// TIA Portal V17 export
// export: Created 2025-03-10T13:12:59.4902027Z, ExportSetting WithDefaults, DisplayName Totally Integrated Automation Portal, DisplayVersion V17 Update 8, DisplayName TIA Portal Openness, DisplayVersion V17 Update 8, DisplayName TIA Portal Version Control Interface, DisplayVersion V17, DisplayName SINAMICS Startdrive Advanced, DisplayVersion V17 SP2, DisplayName SINAMICS Startdrive G110M, G120, G120C, G120D, G120P, G115D, DisplayVersion V17 SP2, DisplayName SINAMICS Startdrive G130, G150, S120, S150, SINAMICS MV, S210, DisplayVersion V17 SP2, DisplayName STEP 7 Professional, DisplayVersion V17 Update 8, DisplayName SINUMERIK ONE STEP 7 Toolbox, DisplayVersion V17 Update 12, DisplayName SINUMERIK 840D sl STEP 7 Toolbox, DisplayVersion V17 Update 12, DisplayName STEP 7 Safety, DisplayVersion V17 Update 6, DisplayName WinCC Advanced, DisplayVersion V17 Update 8
FUNCTION_BLOCK "FB22702_LOAD_FEEDER_SEQUENCE_WEIGHT"   // FB22702, LAD
TITLE = FB22701 LOAD FEEDER SEQUENCE
{ S7_Optimized_Access := 'FALSE' }
VERSION : 0.1
// stored: AutoNumber false, IsIECCheckEnabled false, SetENOAutomatically false, UDAEnableTagReadback false
   VAR_INPUT
      iCONTROL_ON_DELAYED : Bool;
      iPNEUMATIC_FEEDBACK_ON : Bool;
      iFEEDER_PROFINET_MODE_ACTIVE_FAULT : Bool;
      iFEEDER_LINE_NOT_READY_FAULT : Bool;
      iMOTOR_STIRRER_CONDITIONS : Bool;
      iHOPPER_FEEDBACK_PRESSURE : Real;
      iHOPPER_MOTOR_STIRRER_FEEDBACK_SPEED : Real;
      iPOWDER_FEEDER_HOPPER_FEEDBACK_PRESSURE : Real;
      iHOPPER_WEIGHT_FEEDBACK : Real;
      iTRANSFER_VALVE_FEEDBACK_ON : Bool;
      iTRANSFER_VALVE_FEEDBACK_OFF : Bool;
      iPOWDER_FLOW_ON : Bool;
      iSTART_MANUAL_REQUEST : Bool;
      iSTART_SEMI_REQUEST : Bool;
      iSTART_AUTO_REQUEST : Bool;
      iSTOP_MANUAL_REQUEST : Bool;
      iSTOP_SEMI_REQUEST : Bool;
      iSTOP_AUTO_REQUEST : Bool;
   END_VAR
   VAR_OUTPUT
      oEXCEEDED_TIME_ALARM : Bool;
      oOUT_OF_RANGE_ALARM : Bool;
      oLOST_CONDITIONS : Bool;
      oIS_ALARMS : Bool;
   END_VAR
   VAR_IN_OUT
      MOTOR_STIRRER_SETPOINT : DInt;   // MOTOR STIRRER SETPOINT
      PRESSURE_SETPOINT : Real;   // PRESSURE SETPOINT
   END_VAR
   VAR DB_SPECIFIC
      DATA_SEQUENCE : "GENERAL_DATA_SEQUENCES";
      HMI_STANDARD : "HMI_DATA_START_STOP";
      INPUT_SETTINGS : Struct
         UNIT_NUMBER : Int;
         HOPPER_NUMBER : Int;
      END_STRUCT;
      HMI_SEQUENCE : Struct
         HMI_SEQUENCE_RUNNING : Bool;
         HMI_SEQUENCE_DONE : Bool;
         HMI_SET_KILOGRAMS : UDInt;
         HMI_FEEDBACK_DEPOSITED_KG : UDInt;
         HMI_PRESSURE_INCREMENT : Real;
      END_STRUCT;
      ACTIONS_SEQUENCE : Struct
         REQ_START_TRANSFER_POWDER_VALVE : Bool;   // REQUEST OPEN TRANSFER POWDER VALVE
         REQ_STOP_TRANSFER_POWDER_VALVE : Bool;   // REQUEST CLOSE TRANSFER POWDER VALVE
         REQ_START_PRESSURE_GAS_CONTROL : Bool;   // REQUEST START PRESSURE GAS CONTROL
         REQ_STOP_PRESSURE_GAS_CONTROL : Bool;   // REQUEST STOP PRESSURE GAS CONTROL
         REQ_START_PRESSURE_GAS_VALVE : Bool;   // REQUEST OPEN PRESSURE GAS VALVE
         REQ_STOP_PRESSURE_GAS_VALVE : Bool;   // REQUEST CLOSE PRESSURE GAS VALVE
         REQ_START_RELIEF_GAS_VALVE : Bool;   // REQUEST OPEN RELIEF GAS VALVE
         REQ_STOP_RELIEF_GAS_VALVE : Bool;   // REQUEST CLOSE RELIEF GAS VALVE
         SETPOINT_PRESSURE : Real;   // PRESSURE SETPOINT
         REQUEST_START_MOTOR_STIRRER : Bool;   // REQUEST START MOTOR STIRRER
         REQUEST_STOP_MOTOR_STIRRER : Bool;   // REQUEST STOP MOTOR STIRRER
         SETPOINT_MOTOR_STIRRER : DInt;   // MOTOR STIRRER SETPOINT
      END_STRUCT;
      CONTROL_SEQUENCE : Struct
         HOPPER_PRESSURE_IN_RANGE : Bool;
         HOPPER_MOTOR_STIRRER_IN_RANGE : Bool;
         HOPPER_STIRRER_LOW_RANGE : DInt;
         HOPPER_STIRRER_HIGH_RANGE : DInt;
         HOPPER_PRESSURE_LOW_RANGE : Real;
         HOPPER_PRESSURE_HIGH_RANGE : Real;
         HOPPER_PRESSURE_INCREMENT : Real;
         MATERIAL_APPLIED : Bool;
         WEIGHT_APPLIED : UDInt;
         INITIAL_WEIGHT : Real;
         ESTIMATED_WEIGHT_TO_STOP : Real;
      END_STRUCT;
      INTERNAL : Struct
         TRIGGER_RAISING_EDGE_1 : Bool;
         TRIGGER_RAISING_EDGE_2 : Bool;
         TRIGGER_RAISING_EDGE_3 : Bool;
      END_STRUCT;
      TIMERS : Struct
         TIMER_1 : TON_TIME;
         TIMER_2 : TON_TIME;
         TIMER_3 : TON_TIME;
         TIMER_4 : TON_TIME;
         TIMER_5 : TON_TIME;
         TIMER_6 : TON_TIME;
         TIMER_7 : TON_TIME;
         TIMER_8 : TON_TIME;
         TIMER_9 : TON_TIME;
         TIMER_10 : TON_TIME;
      END_STRUCT;
   END_VAR
   VAR_TEMP
      DB_NUMBER : DInt;
      FEEDER_COVER_PRESSURE_ADDED : Real;
      TIME_EXCEEDED_S5TIME : S5Time;
      TIME_COUNTED : Int;
      TIME_EXCEEDED_TIME : Time;
      TIME_LOAD_IN_MILISEC : Int;
      REMAINING_TIME : Int;
      UINT_TIME_ACTION : UInt;
      LOW_FEEDBACK_PRESSURE : Real;
      HIGH_FEEDBACK_PRESSURE : Real;
      LOW_FEEDBACK_MOTOR_SPEED : Real;
      HIGH_FEEDBACK_MOTOR_SPEED : Real;
   END_VAR
   VAR CONSTANT
      HISTERESIS_PRESSURE : Real := 0.04;
   END_VAR
   // TIMERS.TIMER_1.PT := T#1000ms;
   // TIMERS.TIMER_2.PT := T#1000ms;
   // TIMERS.TIMER_3.PT := T#1000ms;
   // TIMERS.TIMER_4.PT := T#1000ms;
   // TIMERS.TIMER_5.PT := T#1000ms;
   // TIMERS.TIMER_6.PT := T#1000ms;
   // TIMERS.TIMER_7.PT := T#1000ms;
   // TIMERS.TIMER_8.PT := T#1000ms;
   // TIMERS.TIMER_9.PT := T#1000ms;
   VAR_TEMP   // added for the SCL form of the ladder/FBD networks
      _w1 : Bool;
      _w2 : Bool;
   END_VAR
BEGIN

NETWORK
TITLE = READ INSTANCE DB NUMBER
      L     DINO;
      +     10#800000;
      T     #DB_NUMBER;

REGION Network 2: INPUTS
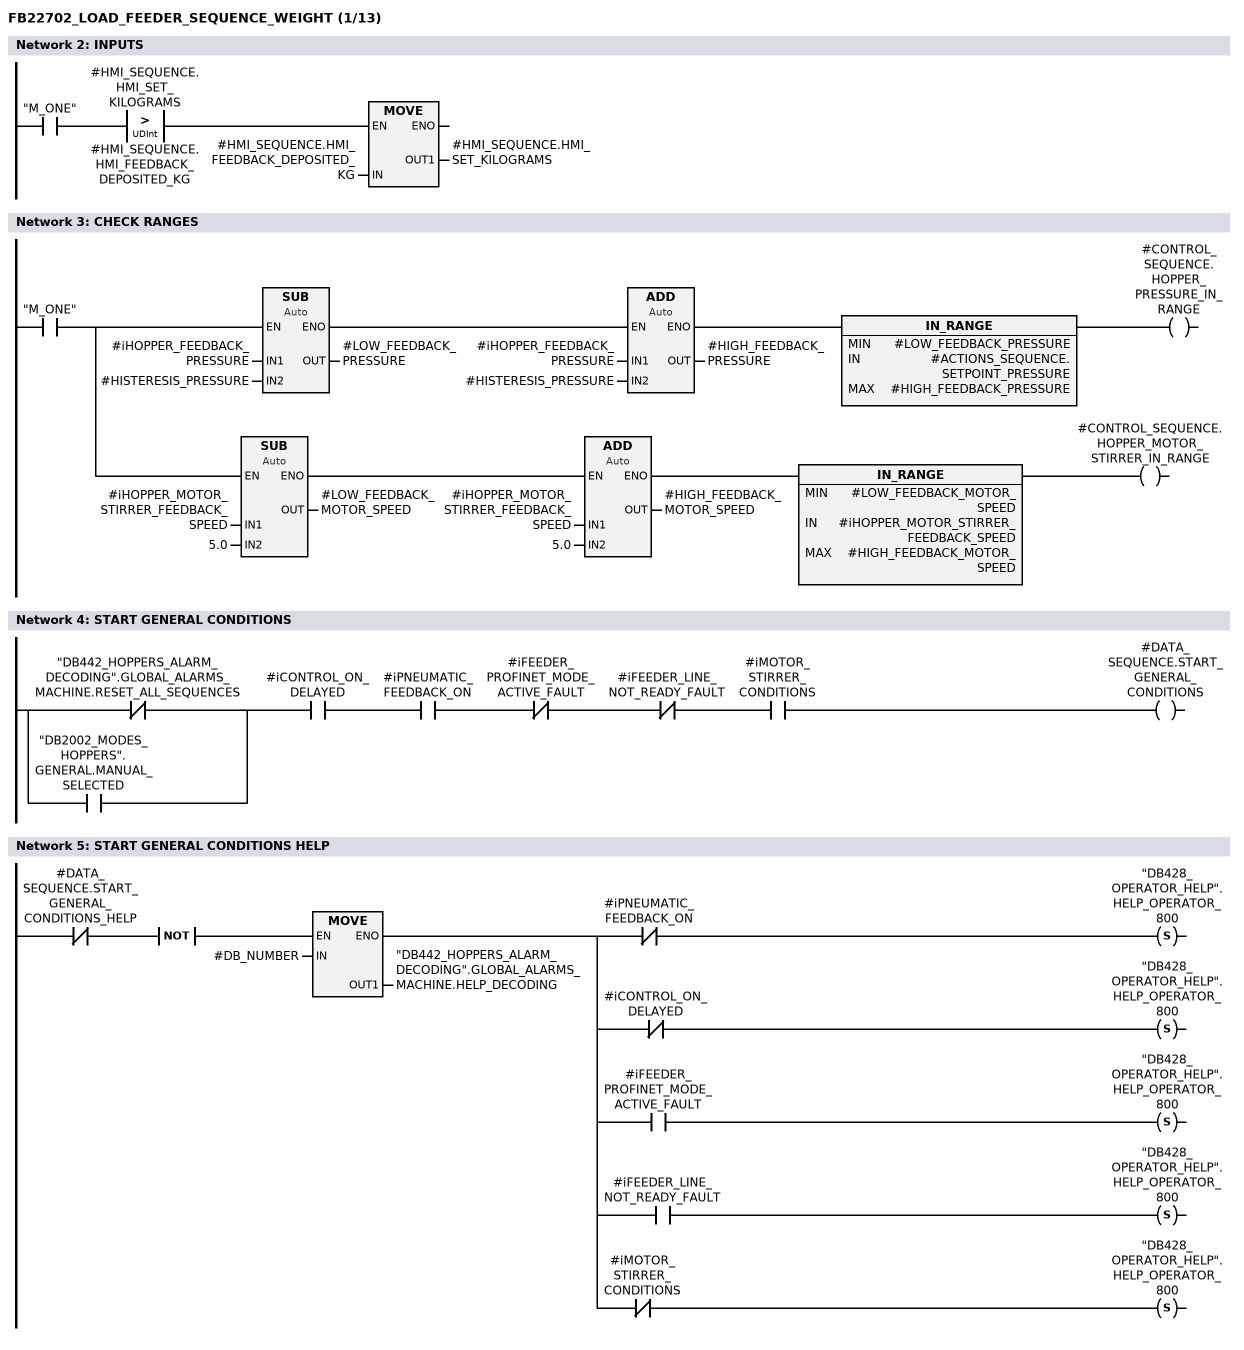
   RUNG wire#powerrail
      Contact( "M_ONE" )
      { S7_Templates := "SrcType := UDInt" } GT_Contact(in1 := #HMI_SEQUENCE.HMI_SET_KILOGRAMS, in2 := #HMI_SEQUENCE.HMI_FEEDBACK_DEPOSITED_KG)
      Move(in := #HMI_SEQUENCE.HMI_FEEDBACK_DEPOSITED_KG, out1 => #HMI_SEQUENCE.HMI_SET_KILOGRAMS)
   END_RUNG
   // the same network as SCL:
   IF "M_ONE" AND (#HMI_SEQUENCE.HMI_SET_KILOGRAMS > #HMI_SEQUENCE.HMI_FEEDBACK_DEPOSITED_KG) THEN
       #HMI_SEQUENCE.HMI_SET_KILOGRAMS := #HMI_SEQUENCE.HMI_FEEDBACK_DEPOSITED_KG;
   END_IF;
END_REGION

REGION Network 3: CHECK RANGES
   RUNG wire#powerrail
      Contact( "M_ONE" )
      wire#w1
      Sub(in1 := #iHOPPER_FEEDBACK_PRESSURE, in2 := #HISTERESIS_PRESSURE, out => #LOW_FEEDBACK_PRESSURE)
      Add(in1 := #iHOPPER_FEEDBACK_PRESSURE, in2 := #HISTERESIS_PRESSURE, out => #HIGH_FEEDBACK_PRESSURE)
      { S7_Templates := "SrcType := Real" } InRange(min := #LOW_FEEDBACK_PRESSURE, in := #ACTIONS_SEQUENCE.SETPOINT_PRESSURE, max := #HIGH_FEEDBACK_PRESSURE)
      Coil( #CONTROL_SEQUENCE.HOPPER_PRESSURE_IN_RANGE )
   END_RUNG
   RUNG wire#w1
      Sub(in1 := #iHOPPER_MOTOR_STIRRER_FEEDBACK_SPEED, in2 := 5.0, out => #LOW_FEEDBACK_MOTOR_SPEED)
      Add(in1 := #iHOPPER_MOTOR_STIRRER_FEEDBACK_SPEED, in2 := 5.0, out => #HIGH_FEEDBACK_MOTOR_SPEED)
      { S7_Templates := "SrcType := Real" } InRange(min := #LOW_FEEDBACK_MOTOR_SPEED, in := #iHOPPER_MOTOR_STIRRER_FEEDBACK_SPEED, max := #HIGH_FEEDBACK_MOTOR_SPEED)
      Coil( #CONTROL_SEQUENCE.HOPPER_MOTOR_STIRRER_IN_RANGE )
   END_RUNG
   // the same network as SCL:
   IF "M_ONE" THEN
       #LOW_FEEDBACK_PRESSURE := #iHOPPER_FEEDBACK_PRESSURE - #HISTERESIS_PRESSURE;
       #HIGH_FEEDBACK_PRESSURE := #iHOPPER_FEEDBACK_PRESSURE + #HISTERESIS_PRESSURE;
   END_IF;
   #CONTROL_SEQUENCE.HOPPER_PRESSURE_IN_RANGE := "M_ONE" AND (#LOW_FEEDBACK_PRESSURE <= #ACTIONS_SEQUENCE.SETPOINT_PRESSURE) AND (#ACTIONS_SEQUENCE.SETPOINT_PRESSURE <= #HIGH_FEEDBACK_PRESSURE);
   IF "M_ONE" THEN
       #LOW_FEEDBACK_MOTOR_SPEED := #iHOPPER_MOTOR_STIRRER_FEEDBACK_SPEED - 5.0;
       #HIGH_FEEDBACK_MOTOR_SPEED := #iHOPPER_MOTOR_STIRRER_FEEDBACK_SPEED + 5.0;
   END_IF;
   #CONTROL_SEQUENCE.HOPPER_MOTOR_STIRRER_IN_RANGE := "M_ONE" AND (#LOW_FEEDBACK_MOTOR_SPEED <= #iHOPPER_MOTOR_STIRRER_FEEDBACK_SPEED) AND (#iHOPPER_MOTOR_STIRRER_FEEDBACK_SPEED <= #HIGH_FEEDBACK_MOTOR_SPEED);
END_REGION

REGION Network 4: START GENERAL CONDITIONS
   RUNG wire#powerrail
      I_Contact( "DB442_HOPPERS_ALARM_DECODING".GLOBAL_ALARMS_MACHINE.RESET_ALL_SEQUENCES )
      wire#w1
      Contact( #iCONTROL_ON_DELAYED )
      Contact( #iPNEUMATIC_FEEDBACK_ON )
      I_Contact( #iFEEDER_PROFINET_MODE_ACTIVE_FAULT )
      I_Contact( #iFEEDER_LINE_NOT_READY_FAULT )
      Contact( #iMOTOR_STIRRER_CONDITIONS )
      Coil( #DATA_SEQUENCE.START_GENERAL_CONDITIONS )
   END_RUNG
   RUNG wire#powerrail
      Contact( "DB2002_MODES_HOPPERS".GENERAL.MANUAL_SELECTED )
   END_RUNG wire#w1
   // the same network as SCL:
   #DATA_SEQUENCE.START_GENERAL_CONDITIONS := (NOT "DB442_HOPPERS_ALARM_DECODING".GLOBAL_ALARMS_MACHINE.RESET_ALL_SEQUENCES OR "DB2002_MODES_HOPPERS".GENERAL.MANUAL_SELECTED) AND #iCONTROL_ON_DELAYED AND #iPNEUMATIC_FEEDBACK_ON AND NOT #iFEEDER_PROFINET_MODE_ACTIVE_FAULT AND NOT #iFEEDER_LINE_NOT_READY_FAULT AND #iMOTOR_STIRRER_CONDITIONS;
END_REGION

REGION Network 5: START GENERAL CONDITIONS HELP
   RUNG wire#powerrail
      I_Contact( #DATA_SEQUENCE.START_GENERAL_CONDITIONS_HELP )
      Not()
      Move(in := #DB_NUMBER, out1 => "DB442_HOPPERS_ALARM_DECODING".GLOBAL_ALARMS_MACHINE.HELP_DECODING)
      wire#w1
      I_Contact( #iPNEUMATIC_FEEDBACK_ON )
      S_Coil( "DB428_OPERATOR_HELP".HELP_OPERATOR_800 )
   END_RUNG
   RUNG wire#w1
      I_Contact( #iCONTROL_ON_DELAYED )
      S_Coil( "DB428_OPERATOR_HELP".HELP_OPERATOR_800 )
   END_RUNG
   RUNG wire#w1
      Contact( #iFEEDER_PROFINET_MODE_ACTIVE_FAULT )
      S_Coil( "DB428_OPERATOR_HELP".HELP_OPERATOR_800 )
   END_RUNG
   RUNG wire#w1
      Contact( #iFEEDER_LINE_NOT_READY_FAULT )
      S_Coil( "DB428_OPERATOR_HELP".HELP_OPERATOR_800 )
   END_RUNG
   RUNG wire#w1
      I_Contact( #iMOTOR_STIRRER_CONDITIONS )
      S_Coil( "DB428_OPERATOR_HELP".HELP_OPERATOR_800 )
   END_RUNG
   // the same network as SCL:
   #_w1 := NOT (NOT #DATA_SEQUENCE.START_GENERAL_CONDITIONS_HELP);
   IF #_w1 THEN "DB442_HOPPERS_ALARM_DECODING".GLOBAL_ALARMS_MACHINE.HELP_DECODING := #DB_NUMBER; END_IF;
   IF #_w1 AND NOT #iPNEUMATIC_FEEDBACK_ON THEN "DB428_OPERATOR_HELP".HELP_OPERATOR_800 := TRUE; END_IF;
   IF #_w1 AND NOT #iCONTROL_ON_DELAYED THEN "DB428_OPERATOR_HELP".HELP_OPERATOR_800 := TRUE; END_IF;
   IF #_w1 AND #iFEEDER_PROFINET_MODE_ACTIVE_FAULT THEN
       "DB428_OPERATOR_HELP".HELP_OPERATOR_800 := TRUE;
   END_IF;
   IF #_w1 AND #iFEEDER_LINE_NOT_READY_FAULT THEN "DB428_OPERATOR_HELP".HELP_OPERATOR_800 := TRUE; END_IF;
   IF #_w1 AND NOT #iMOTOR_STIRRER_CONDITIONS THEN "DB428_OPERATOR_HELP".HELP_OPERATOR_800 := TRUE; END_IF;
END_REGION

REGION Network 6: START INITIAL CONDITIONS / Initial Start Conditions
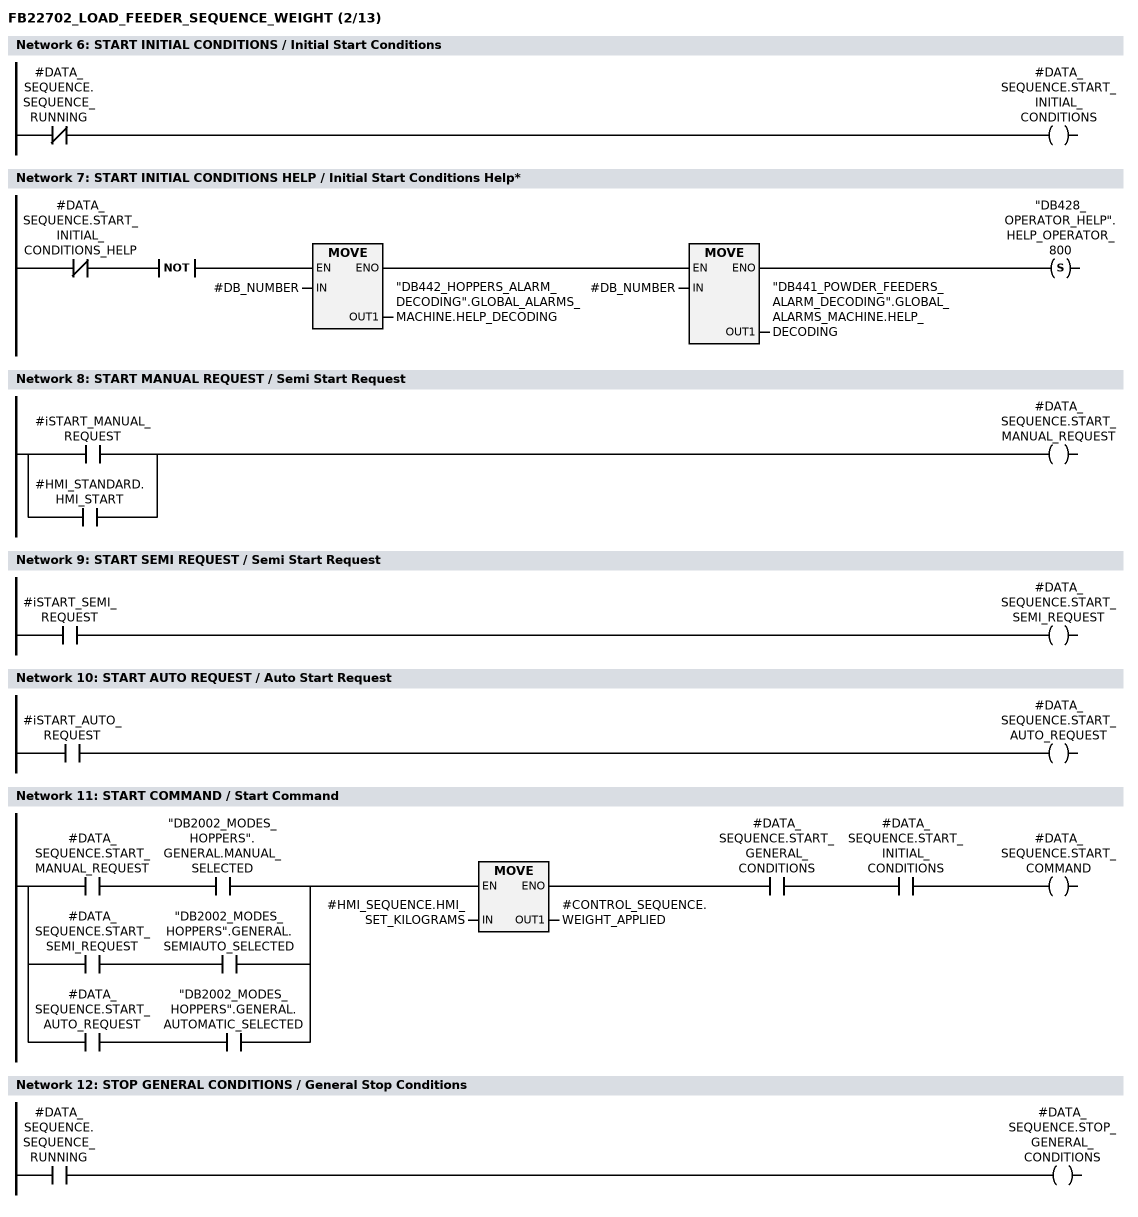
   RUNG wire#powerrail
      I_Contact( #DATA_SEQUENCE.SEQUENCE_RUNNING )
      Coil( #DATA_SEQUENCE.START_INITIAL_CONDITIONS )
   END_RUNG
   // the same network as SCL:
   #DATA_SEQUENCE.START_INITIAL_CONDITIONS := NOT #DATA_SEQUENCE.SEQUENCE_RUNNING;
END_REGION

REGION Network 7: START INITIAL CONDITIONS HELP / Initial Start Conditions Help*
   RUNG wire#powerrail
      I_Contact( #DATA_SEQUENCE.START_INITIAL_CONDITIONS_HELP )
      Not()
      { S7_GenerateENO := "TRUE" } Move(in := #DB_NUMBER, out1 => "DB442_HOPPERS_ALARM_DECODING".GLOBAL_ALARMS_MACHINE.HELP_DECODING)
      { S7_GenerateENO := "TRUE" } Move(in := #DB_NUMBER, out1 => "DB441_POWDER_FEEDERS_ALARM_DECODING".GLOBAL_ALARMS_MACHINE.HELP_DECODING)
      S_Coil( "DB428_OPERATOR_HELP".HELP_OPERATOR_800 )
   END_RUNG
   // the same network as SCL:
   // ENO of a box is taken as its EN; it also drops when the box reports an error
   IF NOT (NOT #DATA_SEQUENCE.START_INITIAL_CONDITIONS_HELP) THEN
       "DB442_HOPPERS_ALARM_DECODING".GLOBAL_ALARMS_MACHINE.HELP_DECODING := #DB_NUMBER;
       "DB441_POWDER_FEEDERS_ALARM_DECODING".GLOBAL_ALARMS_MACHINE.HELP_DECODING := #DB_NUMBER;
       "DB428_OPERATOR_HELP".HELP_OPERATOR_800 := TRUE;
   END_IF;
END_REGION

REGION Network 8: START MANUAL REQUEST / Semi Start Request
   RUNG wire#powerrail
      Contact( #iSTART_MANUAL_REQUEST )
      wire#w1
      Coil( #DATA_SEQUENCE.START_MANUAL_REQUEST )
   END_RUNG
   RUNG wire#powerrail
      Contact( #HMI_STANDARD.HMI_START )
   END_RUNG wire#w1
   // the same network as SCL:
   #DATA_SEQUENCE.START_MANUAL_REQUEST := #iSTART_MANUAL_REQUEST OR #HMI_STANDARD.HMI_START;
END_REGION

REGION Network 9: START SEMI REQUEST / Semi Start Request
   RUNG wire#powerrail
      Contact( #iSTART_SEMI_REQUEST )
      Coil( #DATA_SEQUENCE.START_SEMI_REQUEST )
   END_RUNG
   // the same network as SCL:
   #DATA_SEQUENCE.START_SEMI_REQUEST := #iSTART_SEMI_REQUEST;
END_REGION

REGION Network 10: START AUTO REQUEST / Auto Start Request
   RUNG wire#powerrail
      Contact( #iSTART_AUTO_REQUEST )
      Coil( #DATA_SEQUENCE.START_AUTO_REQUEST )
   END_RUNG
   // the same network as SCL:
   #DATA_SEQUENCE.START_AUTO_REQUEST := #iSTART_AUTO_REQUEST;
END_REGION

REGION Network 11: START COMMAND / Start Command
   RUNG wire#powerrail
      Contact( #DATA_SEQUENCE.START_MANUAL_REQUEST )
      Contact( "DB2002_MODES_HOPPERS".GENERAL.MANUAL_SELECTED )
      wire#w1
      Move(in := #HMI_SEQUENCE.HMI_SET_KILOGRAMS, out1 => #CONTROL_SEQUENCE.WEIGHT_APPLIED)
      Contact( #DATA_SEQUENCE.START_GENERAL_CONDITIONS )
      Contact( #DATA_SEQUENCE.START_INITIAL_CONDITIONS )
      Coil( #DATA_SEQUENCE.START_COMMAND )
   END_RUNG
   RUNG wire#powerrail
      Contact( #DATA_SEQUENCE.START_SEMI_REQUEST )
      Contact( "DB2002_MODES_HOPPERS".GENERAL.SEMIAUTO_SELECTED )
   END_RUNG wire#w1
   RUNG wire#powerrail
      Contact( #DATA_SEQUENCE.START_AUTO_REQUEST )
      Contact( "DB2002_MODES_HOPPERS".GENERAL.AUTOMATIC_SELECTED )
   END_RUNG wire#w1
   // the same network as SCL:
   #_w1 := (#DATA_SEQUENCE.START_MANUAL_REQUEST AND "DB2002_MODES_HOPPERS".GENERAL.MANUAL_SELECTED) OR (#DATA_SEQUENCE.START_SEMI_REQUEST AND "DB2002_MODES_HOPPERS".GENERAL.SEMIAUTO_SELECTED) OR (#DATA_SEQUENCE.START_AUTO_REQUEST AND "DB2002_MODES_HOPPERS".GENERAL.AUTOMATIC_SELECTED);
   IF #_w1 THEN #CONTROL_SEQUENCE.WEIGHT_APPLIED := #HMI_SEQUENCE.HMI_SET_KILOGRAMS; END_IF;
   #DATA_SEQUENCE.START_COMMAND := #_w1 AND #DATA_SEQUENCE.START_GENERAL_CONDITIONS AND #DATA_SEQUENCE.START_INITIAL_CONDITIONS;
END_REGION

REGION Network 12: STOP GENERAL CONDITIONS / General Stop Conditions
   RUNG wire#powerrail
      Contact( #DATA_SEQUENCE.SEQUENCE_RUNNING )
      Coil( #DATA_SEQUENCE.STOP_GENERAL_CONDITIONS )
   END_RUNG
   // the same network as SCL:
   #DATA_SEQUENCE.STOP_GENERAL_CONDITIONS := #DATA_SEQUENCE.SEQUENCE_RUNNING;
END_REGION

REGION Network 13: STOP GENERAL CONDITIONS HELP / General Stop Conditions Help**
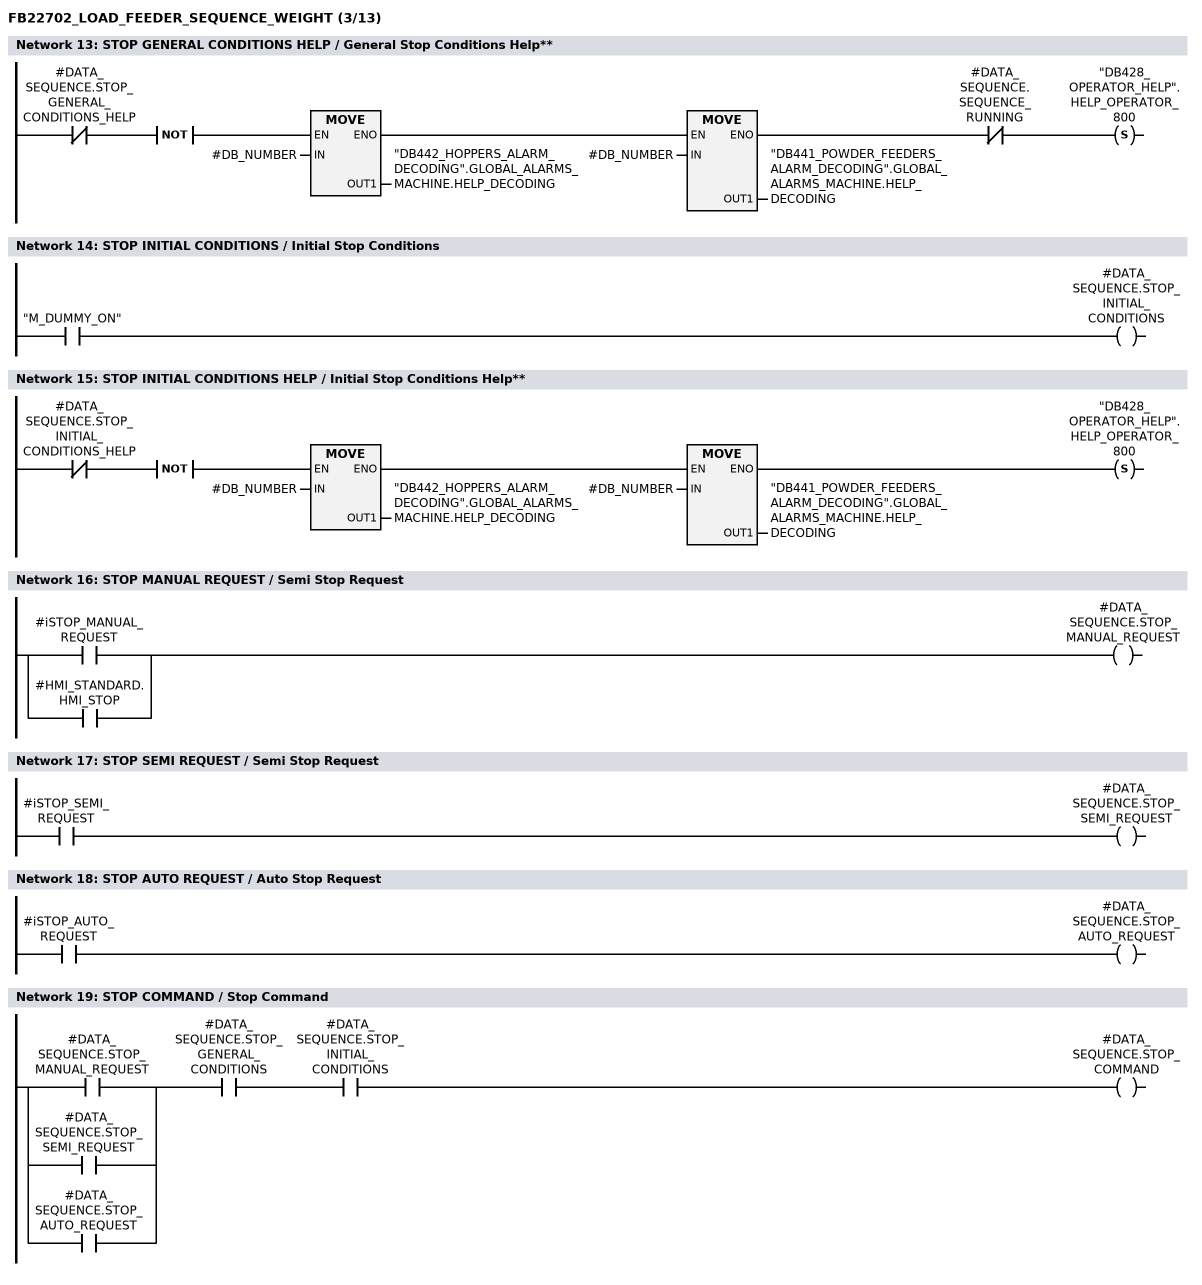
   RUNG wire#powerrail
      I_Contact( #DATA_SEQUENCE.STOP_GENERAL_CONDITIONS_HELP )
      Not()
      { S7_GenerateENO := "TRUE" } Move(in := #DB_NUMBER, out1 => "DB442_HOPPERS_ALARM_DECODING".GLOBAL_ALARMS_MACHINE.HELP_DECODING)
      { S7_GenerateENO := "TRUE" } Move(in := #DB_NUMBER, out1 => "DB441_POWDER_FEEDERS_ALARM_DECODING".GLOBAL_ALARMS_MACHINE.HELP_DECODING)
      I_Contact( #DATA_SEQUENCE.SEQUENCE_RUNNING )
      S_Coil( "DB428_OPERATOR_HELP".HELP_OPERATOR_800 )
   END_RUNG
   // the same network as SCL:
   // ENO of a box is taken as its EN; it also drops when the box reports an error
   #_w1 := NOT (NOT #DATA_SEQUENCE.STOP_GENERAL_CONDITIONS_HELP);
   IF #_w1 THEN
       "DB442_HOPPERS_ALARM_DECODING".GLOBAL_ALARMS_MACHINE.HELP_DECODING := #DB_NUMBER;
       "DB441_POWDER_FEEDERS_ALARM_DECODING".GLOBAL_ALARMS_MACHINE.HELP_DECODING := #DB_NUMBER;
   END_IF;
   IF #_w1 AND NOT #DATA_SEQUENCE.SEQUENCE_RUNNING THEN
       "DB428_OPERATOR_HELP".HELP_OPERATOR_800 := TRUE;
   END_IF;
END_REGION

REGION Network 14: STOP INITIAL CONDITIONS / Initial Stop Conditions
   RUNG wire#powerrail
      Contact( "M_DUMMY_ON" )
      Coil( #DATA_SEQUENCE.STOP_INITIAL_CONDITIONS )
   END_RUNG
   // the same network as SCL:
   #DATA_SEQUENCE.STOP_INITIAL_CONDITIONS := "M_DUMMY_ON";
END_REGION

REGION Network 15: STOP INITIAL CONDITIONS HELP / Initial Stop Conditions Help**
   RUNG wire#powerrail
      I_Contact( #DATA_SEQUENCE.STOP_INITIAL_CONDITIONS_HELP )
      Not()
      { S7_GenerateENO := "TRUE" } Move(in := #DB_NUMBER, out1 => "DB442_HOPPERS_ALARM_DECODING".GLOBAL_ALARMS_MACHINE.HELP_DECODING)
      { S7_GenerateENO := "TRUE" } Move(in := #DB_NUMBER, out1 => "DB441_POWDER_FEEDERS_ALARM_DECODING".GLOBAL_ALARMS_MACHINE.HELP_DECODING)
      S_Coil( "DB428_OPERATOR_HELP".HELP_OPERATOR_800 )
   END_RUNG
   // the same network as SCL:
   // ENO of a box is taken as its EN; it also drops when the box reports an error
   IF NOT (NOT #DATA_SEQUENCE.STOP_INITIAL_CONDITIONS_HELP) THEN
       "DB442_HOPPERS_ALARM_DECODING".GLOBAL_ALARMS_MACHINE.HELP_DECODING := #DB_NUMBER;
       "DB441_POWDER_FEEDERS_ALARM_DECODING".GLOBAL_ALARMS_MACHINE.HELP_DECODING := #DB_NUMBER;
       "DB428_OPERATOR_HELP".HELP_OPERATOR_800 := TRUE;
   END_IF;
END_REGION

REGION Network 16: STOP MANUAL REQUEST / Semi Stop Request
   RUNG wire#powerrail
      Contact( #iSTOP_MANUAL_REQUEST )
      wire#w1
      Coil( #DATA_SEQUENCE.STOP_MANUAL_REQUEST )
   END_RUNG
   RUNG wire#powerrail
      Contact( #HMI_STANDARD.HMI_STOP )
   END_RUNG wire#w1
   // the same network as SCL:
   #DATA_SEQUENCE.STOP_MANUAL_REQUEST := #iSTOP_MANUAL_REQUEST OR #HMI_STANDARD.HMI_STOP;
END_REGION

REGION Network 17: STOP SEMI REQUEST / Semi Stop Request
   RUNG wire#powerrail
      Contact( #iSTOP_SEMI_REQUEST )
      Coil( #DATA_SEQUENCE.STOP_SEMI_REQUEST )
   END_RUNG
   // the same network as SCL:
   #DATA_SEQUENCE.STOP_SEMI_REQUEST := #iSTOP_SEMI_REQUEST;
END_REGION

REGION Network 18: STOP AUTO REQUEST / Auto Stop Request
   RUNG wire#powerrail
      Contact( #iSTOP_AUTO_REQUEST )
      Coil( #DATA_SEQUENCE.STOP_AUTO_REQUEST )
   END_RUNG
   // the same network as SCL:
   #DATA_SEQUENCE.STOP_AUTO_REQUEST := #iSTOP_AUTO_REQUEST;
END_REGION

REGION Network 19: STOP COMMAND / Stop Command
   RUNG wire#powerrail
      Contact( #DATA_SEQUENCE.STOP_MANUAL_REQUEST )
      wire#w1
      Contact( #DATA_SEQUENCE.STOP_GENERAL_CONDITIONS )
      Contact( #DATA_SEQUENCE.STOP_INITIAL_CONDITIONS )
      Coil( #DATA_SEQUENCE.STOP_COMMAND )
   END_RUNG
   RUNG wire#powerrail
      Contact( #DATA_SEQUENCE.STOP_SEMI_REQUEST )
   END_RUNG wire#w1
   RUNG wire#powerrail
      Contact( #DATA_SEQUENCE.STOP_AUTO_REQUEST )
   END_RUNG wire#w1
   // the same network as SCL:
   #DATA_SEQUENCE.STOP_COMMAND := (#DATA_SEQUENCE.STOP_MANUAL_REQUEST OR #DATA_SEQUENCE.STOP_SEMI_REQUEST OR #DATA_SEQUENCE.STOP_AUTO_REQUEST) AND #DATA_SEQUENCE.STOP_GENERAL_CONDITIONS AND #DATA_SEQUENCE.STOP_INITIAL_CONDITIONS;
END_REGION

REGION Network 20: SEQUENCE RUNNING / Sequence Running
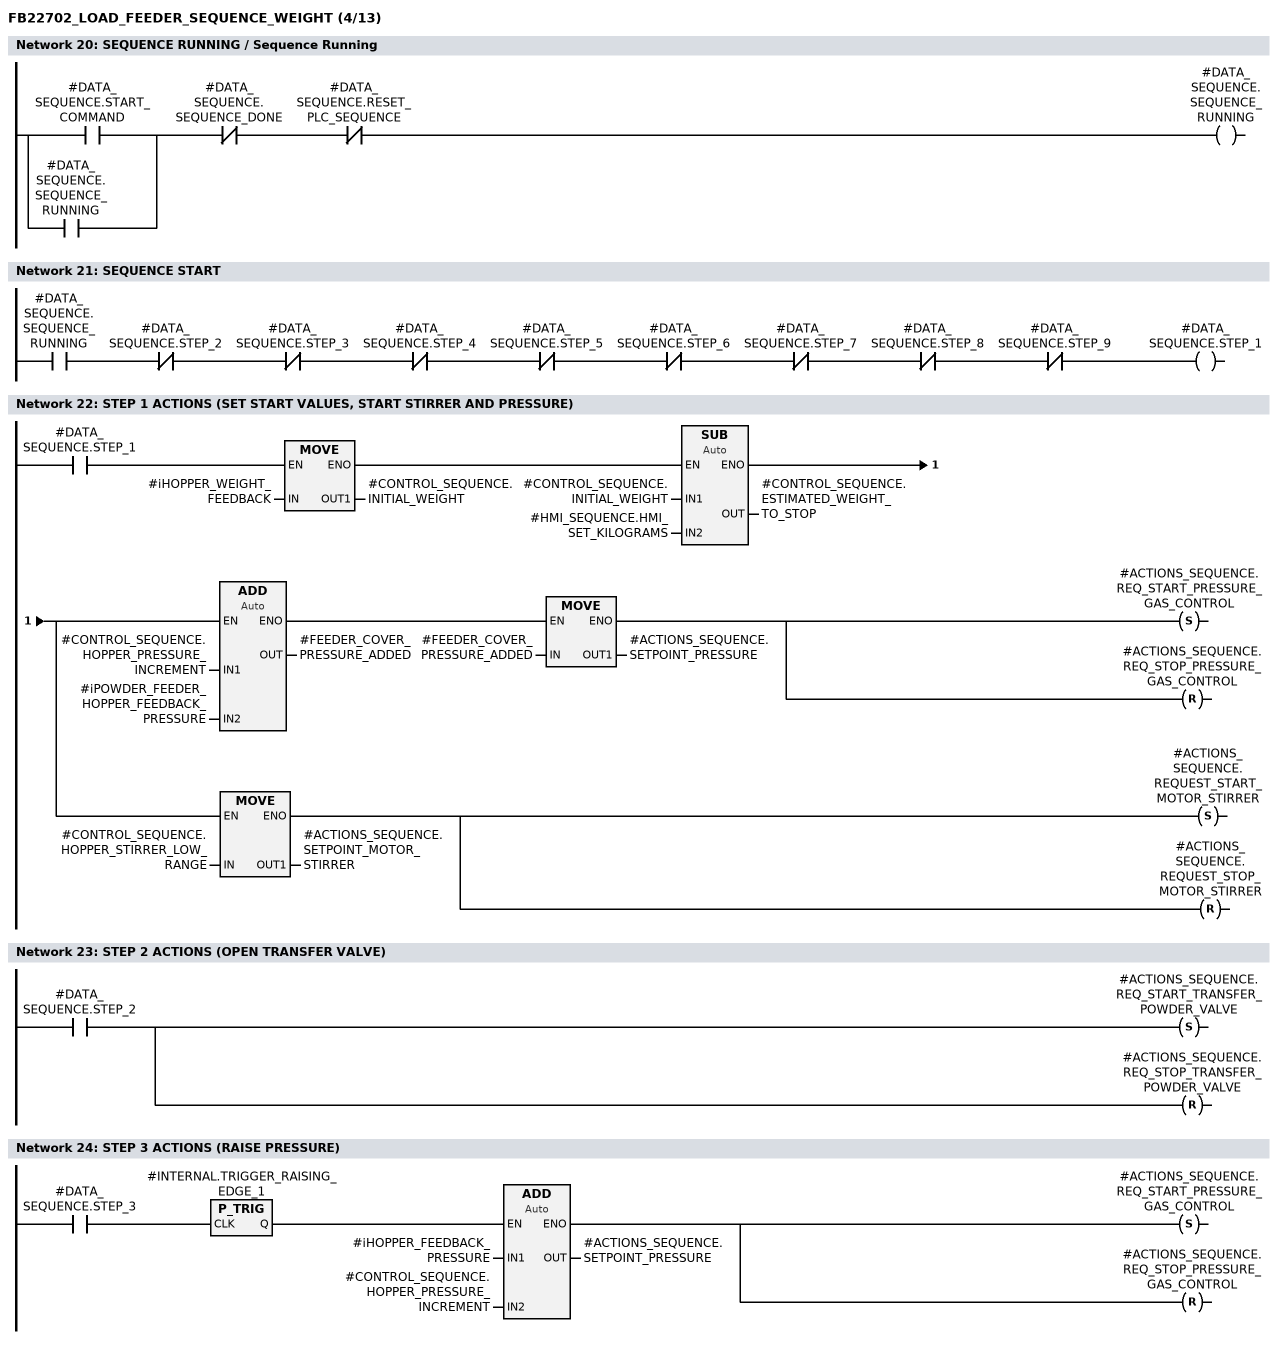
   RUNG wire#powerrail
      Contact( #DATA_SEQUENCE.START_COMMAND )
      wire#w1
      I_Contact( #DATA_SEQUENCE.SEQUENCE_DONE )
      I_Contact( #DATA_SEQUENCE.RESET_PLC_SEQUENCE )
      Coil( #DATA_SEQUENCE.SEQUENCE_RUNNING )
   END_RUNG
   RUNG wire#powerrail
      Contact( #DATA_SEQUENCE.SEQUENCE_RUNNING )
   END_RUNG wire#w1
   // the same network as SCL:
   #DATA_SEQUENCE.SEQUENCE_RUNNING := (#DATA_SEQUENCE.START_COMMAND OR #DATA_SEQUENCE.SEQUENCE_RUNNING) AND NOT #DATA_SEQUENCE.SEQUENCE_DONE AND NOT #DATA_SEQUENCE.RESET_PLC_SEQUENCE;
END_REGION

REGION Network 21: SEQUENCE START
   RUNG wire#powerrail
      Contact( #DATA_SEQUENCE.SEQUENCE_RUNNING )
      I_Contact( #DATA_SEQUENCE.STEP_2 )
      I_Contact( #DATA_SEQUENCE.STEP_3 )
      I_Contact( #DATA_SEQUENCE.STEP_4 )
      I_Contact( #DATA_SEQUENCE.STEP_5 )
      I_Contact( #DATA_SEQUENCE.STEP_6 )
      I_Contact( #DATA_SEQUENCE.STEP_7 )
      I_Contact( #DATA_SEQUENCE.STEP_8 )
      I_Contact( #DATA_SEQUENCE.STEP_9 )
      Coil( #DATA_SEQUENCE.STEP_1 )
   END_RUNG
   // the same network as SCL:
   #DATA_SEQUENCE.STEP_1 := #DATA_SEQUENCE.SEQUENCE_RUNNING AND NOT #DATA_SEQUENCE.STEP_2 AND NOT #DATA_SEQUENCE.STEP_3 AND NOT #DATA_SEQUENCE.STEP_4 AND NOT #DATA_SEQUENCE.STEP_5 AND NOT #DATA_SEQUENCE.STEP_6 AND NOT #DATA_SEQUENCE.STEP_7 AND NOT #DATA_SEQUENCE.STEP_8 AND NOT #DATA_SEQUENCE.STEP_9;
END_REGION

REGION Network 22: STEP 1 ACTIONS (SET START VALUES, START STIRRER AND PRESSURE)
   RUNG wire#powerrail
      Contact( #DATA_SEQUENCE.STEP_1 )
      Move(in := #iHOPPER_WEIGHT_FEEDBACK, out1 => #CONTROL_SEQUENCE.INITIAL_WEIGHT)
      Sub(in1 := #CONTROL_SEQUENCE.INITIAL_WEIGHT, in2 := #HMI_SEQUENCE.HMI_SET_KILOGRAMS, out => #CONTROL_SEQUENCE.ESTIMATED_WEIGHT_TO_STOP)
      wire#w1
      Add(in1 := #CONTROL_SEQUENCE.HOPPER_PRESSURE_INCREMENT, in2 := #iPOWDER_FEEDER_HOPPER_FEEDBACK_PRESSURE, out => #FEEDER_COVER_PRESSURE_ADDED)
      Move(in := #FEEDER_COVER_PRESSURE_ADDED, out1 => #ACTIONS_SEQUENCE.SETPOINT_PRESSURE)
      wire#w2
      S_Coil( #ACTIONS_SEQUENCE.REQ_START_PRESSURE_GAS_CONTROL )
   END_RUNG
   RUNG wire#w2
      R_Coil( #ACTIONS_SEQUENCE.REQ_STOP_PRESSURE_GAS_CONTROL )
   END_RUNG
   RUNG wire#w1
      Move(in := #CONTROL_SEQUENCE.HOPPER_STIRRER_LOW_RANGE, out1 => #ACTIONS_SEQUENCE.SETPOINT_MOTOR_STIRRER)
      wire#w3
      S_Coil( #ACTIONS_SEQUENCE.REQUEST_START_MOTOR_STIRRER )
   END_RUNG
   RUNG wire#w3
      R_Coil( #ACTIONS_SEQUENCE.REQUEST_STOP_MOTOR_STIRRER )
   END_RUNG
   // the same network as SCL:
   IF #DATA_SEQUENCE.STEP_1 THEN
       #CONTROL_SEQUENCE.INITIAL_WEIGHT := #iHOPPER_WEIGHT_FEEDBACK;
       #CONTROL_SEQUENCE.ESTIMATED_WEIGHT_TO_STOP := #CONTROL_SEQUENCE.INITIAL_WEIGHT - #HMI_SEQUENCE.HMI_SET_KILOGRAMS;
       #FEEDER_COVER_PRESSURE_ADDED := #CONTROL_SEQUENCE.HOPPER_PRESSURE_INCREMENT + #iPOWDER_FEEDER_HOPPER_FEEDBACK_PRESSURE;
       #ACTIONS_SEQUENCE.SETPOINT_PRESSURE := #FEEDER_COVER_PRESSURE_ADDED;
       #ACTIONS_SEQUENCE.REQ_START_PRESSURE_GAS_CONTROL := TRUE;
       #ACTIONS_SEQUENCE.REQ_STOP_PRESSURE_GAS_CONTROL := FALSE;
       #ACTIONS_SEQUENCE.SETPOINT_MOTOR_STIRRER := #CONTROL_SEQUENCE.HOPPER_STIRRER_LOW_RANGE;
       #ACTIONS_SEQUENCE.REQUEST_START_MOTOR_STIRRER := TRUE;
       #ACTIONS_SEQUENCE.REQUEST_STOP_MOTOR_STIRRER := FALSE;
   END_IF;
END_REGION

REGION Network 23: STEP 2 ACTIONS (OPEN TRANSFER VALVE)
   RUNG wire#powerrail
      Contact( #DATA_SEQUENCE.STEP_2 )
      wire#w1
      S_Coil( #ACTIONS_SEQUENCE.REQ_START_TRANSFER_POWDER_VALVE )
   END_RUNG
   RUNG wire#w1
      R_Coil( #ACTIONS_SEQUENCE.REQ_STOP_TRANSFER_POWDER_VALVE )
   END_RUNG
   // the same network as SCL:
   IF #DATA_SEQUENCE.STEP_2 THEN
       #ACTIONS_SEQUENCE.REQ_START_TRANSFER_POWDER_VALVE := TRUE;
       #ACTIONS_SEQUENCE.REQ_STOP_TRANSFER_POWDER_VALVE := FALSE;
   END_IF;
END_REGION

REGION Network 24: STEP 3 ACTIONS (RAISE PRESSURE)
   RUNG wire#powerrail
      Contact( #DATA_SEQUENCE.STEP_3 )
      P_Trig( #INTERNAL.TRIGGER_RAISING_EDGE_1 )
      Add(in1 := #iHOPPER_FEEDBACK_PRESSURE, in2 := #CONTROL_SEQUENCE.HOPPER_PRESSURE_INCREMENT, out => #ACTIONS_SEQUENCE.SETPOINT_PRESSURE)
      wire#w1
      S_Coil( #ACTIONS_SEQUENCE.REQ_START_PRESSURE_GAS_CONTROL )
   END_RUNG
   RUNG wire#w1
      R_Coil( #ACTIONS_SEQUENCE.REQ_STOP_PRESSURE_GAS_CONTROL )
   END_RUNG
   // the same network as SCL:
   #_w1 := #DATA_SEQUENCE.STEP_3 AND NOT #INTERNAL.TRIGGER_RAISING_EDGE_1;   // rising edge
   #INTERNAL.TRIGGER_RAISING_EDGE_1 := #DATA_SEQUENCE.STEP_3;
   IF #_w1 THEN
       #ACTIONS_SEQUENCE.SETPOINT_PRESSURE := #iHOPPER_FEEDBACK_PRESSURE + #CONTROL_SEQUENCE.HOPPER_PRESSURE_INCREMENT;
       #ACTIONS_SEQUENCE.REQ_START_PRESSURE_GAS_CONTROL := TRUE;
       #ACTIONS_SEQUENCE.REQ_STOP_PRESSURE_GAS_CONTROL := FALSE;
   END_IF;
END_REGION

REGION Network 25: STEP 4 ACTIONS (RAISE MOTOR SPEED)
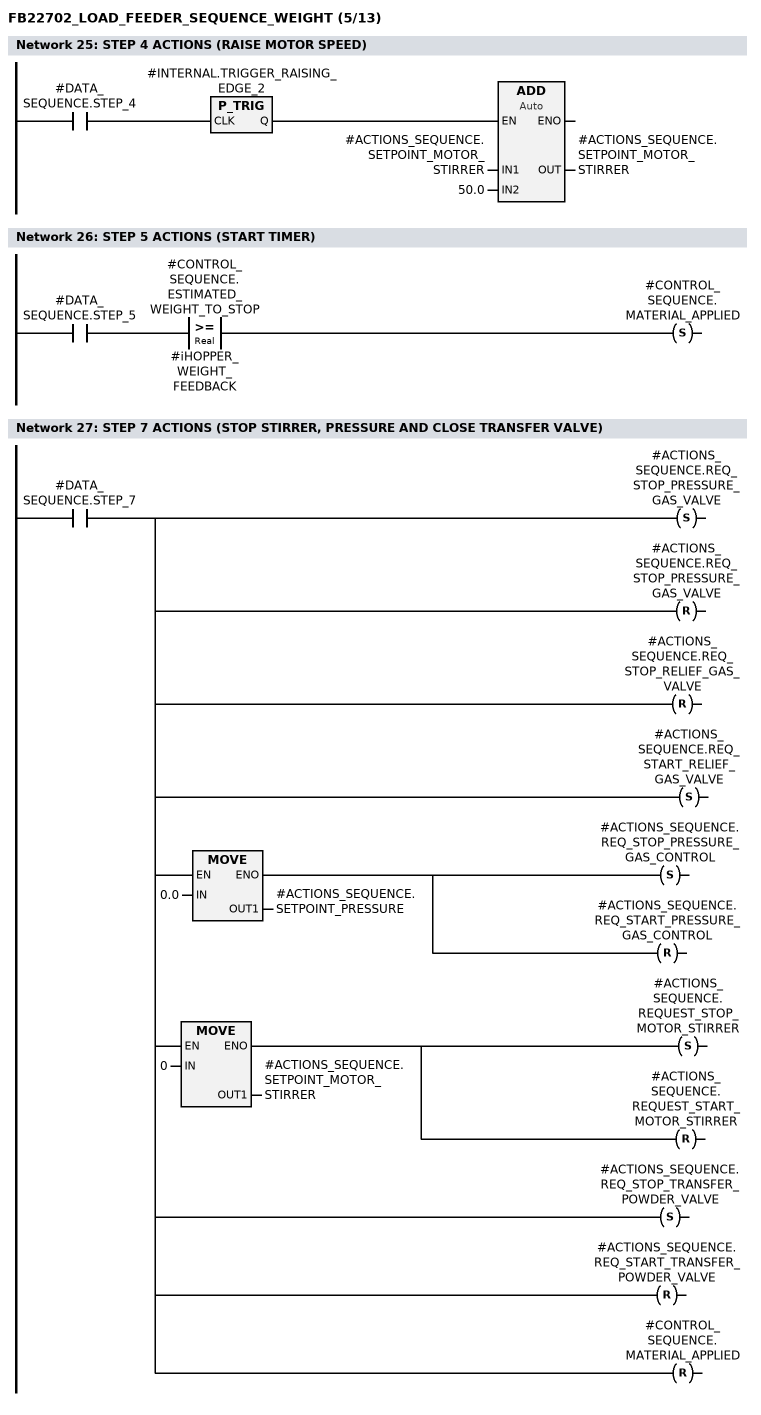
   RUNG wire#powerrail
      Contact( #DATA_SEQUENCE.STEP_4 )
      P_Trig( #INTERNAL.TRIGGER_RAISING_EDGE_2 )
      Add(in1 := #ACTIONS_SEQUENCE.SETPOINT_MOTOR_STIRRER, in2 := 50.0, out => #ACTIONS_SEQUENCE.SETPOINT_MOTOR_STIRRER)
   END_RUNG
   // the same network as SCL:
   #_w1 := #DATA_SEQUENCE.STEP_4 AND NOT #INTERNAL.TRIGGER_RAISING_EDGE_2;   // rising edge
   #INTERNAL.TRIGGER_RAISING_EDGE_2 := #DATA_SEQUENCE.STEP_4;
   IF #_w1 THEN
       #ACTIONS_SEQUENCE.SETPOINT_MOTOR_STIRRER := #ACTIONS_SEQUENCE.SETPOINT_MOTOR_STIRRER + 50.0;
   END_IF;
END_REGION

REGION Network 26: STEP 5 ACTIONS (START TIMER)
   RUNG wire#powerrail
      Contact( #DATA_SEQUENCE.STEP_5 )
      { S7_Templates := "SrcType := Real" } GE_Contact(in1 := #CONTROL_SEQUENCE.ESTIMATED_WEIGHT_TO_STOP, in2 := #iHOPPER_WEIGHT_FEEDBACK)
      S_Coil( #CONTROL_SEQUENCE.MATERIAL_APPLIED )
   END_RUNG
   // the same network as SCL:
   IF #DATA_SEQUENCE.STEP_5 AND (#CONTROL_SEQUENCE.ESTIMATED_WEIGHT_TO_STOP >= #iHOPPER_WEIGHT_FEEDBACK) THEN
       #CONTROL_SEQUENCE.MATERIAL_APPLIED := TRUE;
   END_IF;
END_REGION

REGION Network 27: STEP 7 ACTIONS (STOP STIRRER, PRESSURE AND CLOSE TRANSFER VALVE)
   RUNG wire#powerrail
      Contact( #DATA_SEQUENCE.STEP_7 )
      wire#w1
      S_Coil( #ACTIONS_SEQUENCE.REQ_STOP_PRESSURE_GAS_VALVE )
   END_RUNG
   RUNG wire#w1
      R_Coil( #ACTIONS_SEQUENCE.REQ_STOP_PRESSURE_GAS_VALVE )
   END_RUNG
   RUNG wire#w1
      R_Coil( #ACTIONS_SEQUENCE.REQ_STOP_RELIEF_GAS_VALVE )
   END_RUNG
   RUNG wire#w1
      S_Coil( #ACTIONS_SEQUENCE.REQ_START_RELIEF_GAS_VALVE )
   END_RUNG
   RUNG wire#w1
      Move(in := 0.0, out1 => #ACTIONS_SEQUENCE.SETPOINT_PRESSURE)
      wire#w2
      S_Coil( #ACTIONS_SEQUENCE.REQ_STOP_PRESSURE_GAS_CONTROL )
   END_RUNG
   RUNG wire#w2
      R_Coil( #ACTIONS_SEQUENCE.REQ_START_PRESSURE_GAS_CONTROL )
   END_RUNG
   RUNG wire#w1
      Move(in := 0, out1 => #ACTIONS_SEQUENCE.SETPOINT_MOTOR_STIRRER)
      wire#w3
      S_Coil( #ACTIONS_SEQUENCE.REQUEST_STOP_MOTOR_STIRRER )
   END_RUNG
   RUNG wire#w3
      R_Coil( #ACTIONS_SEQUENCE.REQUEST_START_MOTOR_STIRRER )
   END_RUNG
   RUNG wire#w1
      S_Coil( #ACTIONS_SEQUENCE.REQ_STOP_TRANSFER_POWDER_VALVE )
   END_RUNG
   RUNG wire#w1
      R_Coil( #ACTIONS_SEQUENCE.REQ_START_TRANSFER_POWDER_VALVE )
   END_RUNG
   RUNG wire#w1
      R_Coil( #CONTROL_SEQUENCE.MATERIAL_APPLIED )
   END_RUNG
   // the same network as SCL:
   IF #DATA_SEQUENCE.STEP_7 THEN
       #ACTIONS_SEQUENCE.REQ_STOP_PRESSURE_GAS_VALVE := TRUE;
       #ACTIONS_SEQUENCE.REQ_STOP_PRESSURE_GAS_VALVE := FALSE;
       #ACTIONS_SEQUENCE.REQ_STOP_RELIEF_GAS_VALVE := FALSE;
       #ACTIONS_SEQUENCE.REQ_START_RELIEF_GAS_VALVE := TRUE;
       #ACTIONS_SEQUENCE.SETPOINT_PRESSURE := 0.0;
       #ACTIONS_SEQUENCE.REQ_STOP_PRESSURE_GAS_CONTROL := TRUE;
       #ACTIONS_SEQUENCE.REQ_START_PRESSURE_GAS_CONTROL := FALSE;
       #ACTIONS_SEQUENCE.SETPOINT_MOTOR_STIRRER := 0;
       #ACTIONS_SEQUENCE.REQUEST_STOP_MOTOR_STIRRER := TRUE;
       #ACTIONS_SEQUENCE.REQUEST_START_MOTOR_STIRRER := FALSE;
       #ACTIONS_SEQUENCE.REQ_STOP_TRANSFER_POWDER_VALVE := TRUE;
       #ACTIONS_SEQUENCE.REQ_START_TRANSFER_POWDER_VALVE := FALSE;
       #CONTROL_SEQUENCE.MATERIAL_APPLIED := FALSE;
   END_IF;
END_REGION

REGION Network 28: STEP 8 ACTIONS(STOP STIRRER, PRESSURE AND CLOSE TRANSFER VALVE)
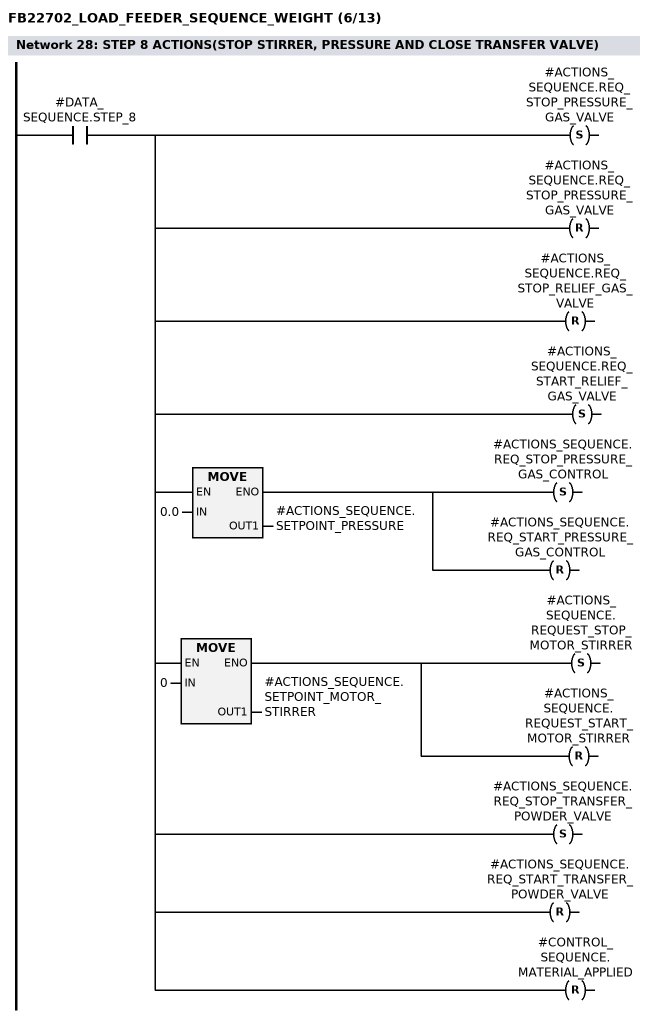
   RUNG wire#powerrail
      Contact( #DATA_SEQUENCE.STEP_8 )
      wire#w1
      S_Coil( #ACTIONS_SEQUENCE.REQ_STOP_PRESSURE_GAS_VALVE )
   END_RUNG
   RUNG wire#w1
      R_Coil( #ACTIONS_SEQUENCE.REQ_STOP_PRESSURE_GAS_VALVE )
   END_RUNG
   RUNG wire#w1
      R_Coil( #ACTIONS_SEQUENCE.REQ_STOP_RELIEF_GAS_VALVE )
   END_RUNG
   RUNG wire#w1
      S_Coil( #ACTIONS_SEQUENCE.REQ_START_RELIEF_GAS_VALVE )
   END_RUNG
   RUNG wire#w1
      Move(in := 0.0, out1 => #ACTIONS_SEQUENCE.SETPOINT_PRESSURE)
      wire#w2
      S_Coil( #ACTIONS_SEQUENCE.REQ_STOP_PRESSURE_GAS_CONTROL )
   END_RUNG
   RUNG wire#w2
      R_Coil( #ACTIONS_SEQUENCE.REQ_START_PRESSURE_GAS_CONTROL )
   END_RUNG
   RUNG wire#w1
      Move(in := 0, out1 => #ACTIONS_SEQUENCE.SETPOINT_MOTOR_STIRRER)
      wire#w3
      S_Coil( #ACTIONS_SEQUENCE.REQUEST_STOP_MOTOR_STIRRER )
   END_RUNG
   RUNG wire#w3
      R_Coil( #ACTIONS_SEQUENCE.REQUEST_START_MOTOR_STIRRER )
   END_RUNG
   RUNG wire#w1
      S_Coil( #ACTIONS_SEQUENCE.REQ_STOP_TRANSFER_POWDER_VALVE )
   END_RUNG
   RUNG wire#w1
      R_Coil( #ACTIONS_SEQUENCE.REQ_START_TRANSFER_POWDER_VALVE )
   END_RUNG
   RUNG wire#w1
      R_Coil( #CONTROL_SEQUENCE.MATERIAL_APPLIED )
   END_RUNG
   // the same network as SCL:
   IF #DATA_SEQUENCE.STEP_8 THEN
       #ACTIONS_SEQUENCE.REQ_STOP_PRESSURE_GAS_VALVE := TRUE;
       #ACTIONS_SEQUENCE.REQ_STOP_PRESSURE_GAS_VALVE := FALSE;
       #ACTIONS_SEQUENCE.REQ_STOP_RELIEF_GAS_VALVE := FALSE;
       #ACTIONS_SEQUENCE.REQ_START_RELIEF_GAS_VALVE := TRUE;
       #ACTIONS_SEQUENCE.SETPOINT_PRESSURE := 0.0;
       #ACTIONS_SEQUENCE.REQ_STOP_PRESSURE_GAS_CONTROL := TRUE;
       #ACTIONS_SEQUENCE.REQ_START_PRESSURE_GAS_CONTROL := FALSE;
       #ACTIONS_SEQUENCE.SETPOINT_MOTOR_STIRRER := 0;
       #ACTIONS_SEQUENCE.REQUEST_STOP_MOTOR_STIRRER := TRUE;
       #ACTIONS_SEQUENCE.REQUEST_START_MOTOR_STIRRER := FALSE;
       #ACTIONS_SEQUENCE.REQ_STOP_TRANSFER_POWDER_VALVE := TRUE;
       #ACTIONS_SEQUENCE.REQ_START_TRANSFER_POWDER_VALVE := FALSE;
       #CONTROL_SEQUENCE.MATERIAL_APPLIED := FALSE;
   END_IF;
END_REGION

REGION Network 29: STEP 9 ACTIONS (RESET VARIABLES)
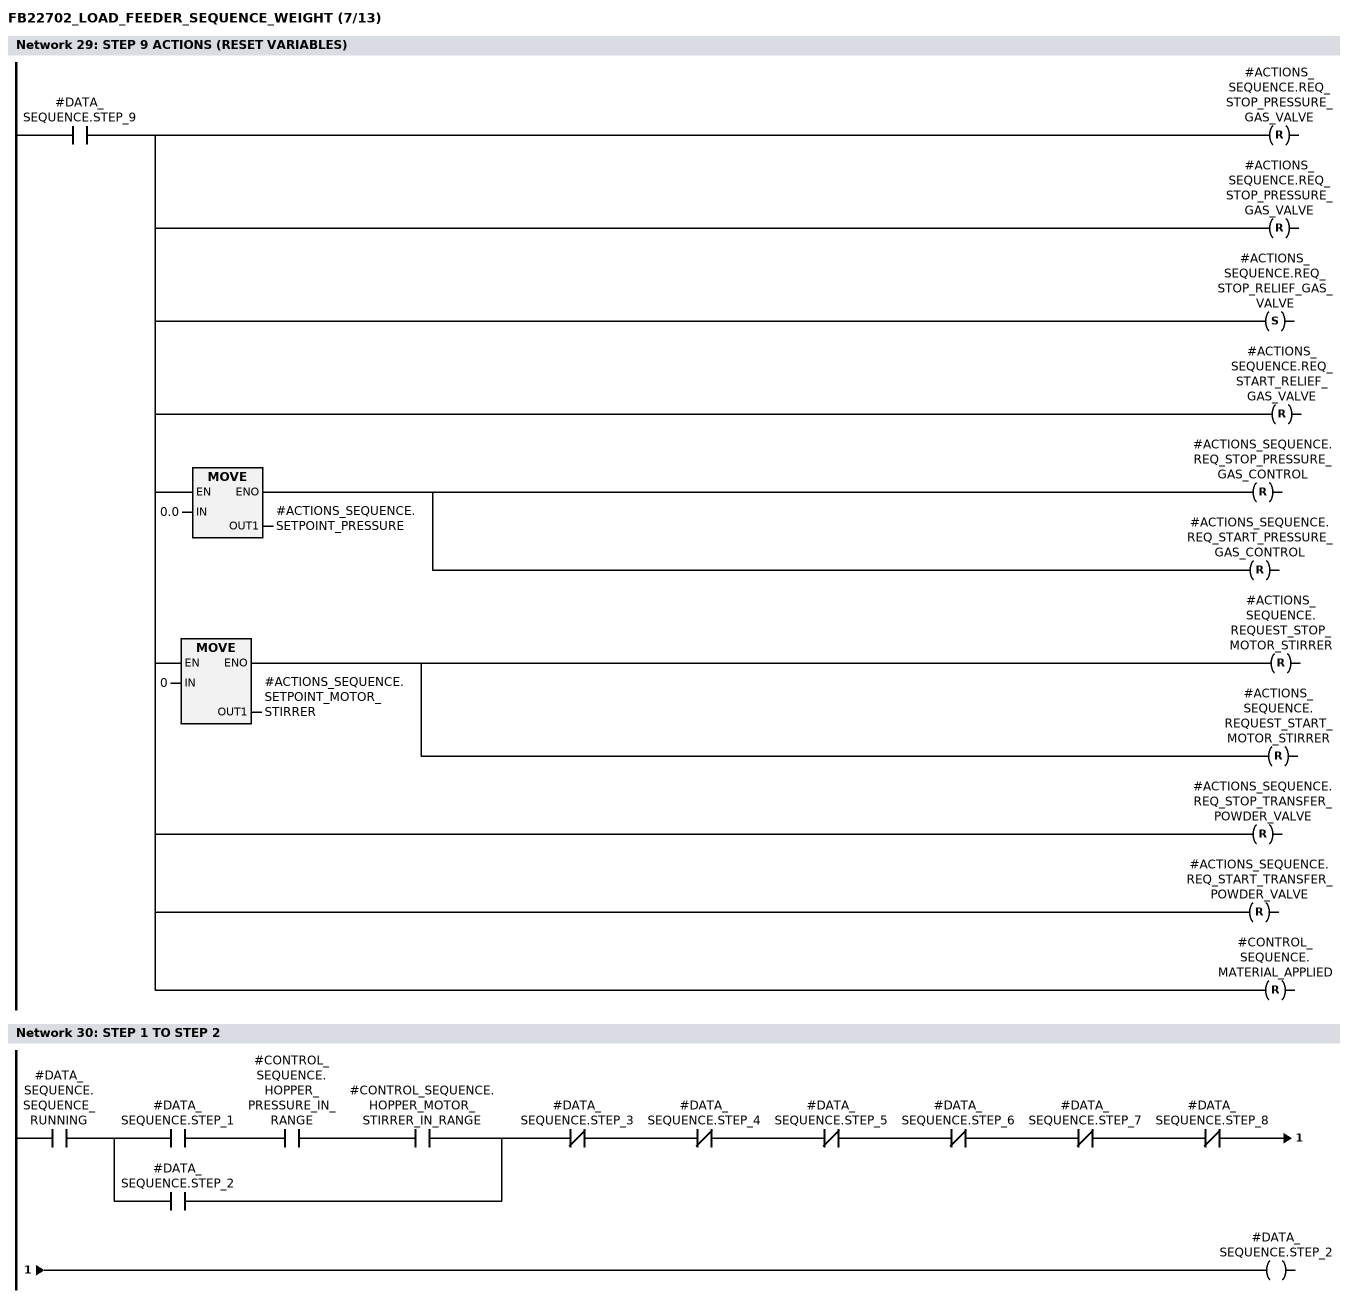
   RUNG wire#powerrail
      Contact( #DATA_SEQUENCE.STEP_9 )
      wire#w1
      R_Coil( #ACTIONS_SEQUENCE.REQ_STOP_PRESSURE_GAS_VALVE )
   END_RUNG
   RUNG wire#w1
      R_Coil( #ACTIONS_SEQUENCE.REQ_STOP_PRESSURE_GAS_VALVE )
   END_RUNG
   RUNG wire#w1
      S_Coil( #ACTIONS_SEQUENCE.REQ_STOP_RELIEF_GAS_VALVE )
   END_RUNG
   RUNG wire#w1
      R_Coil( #ACTIONS_SEQUENCE.REQ_START_RELIEF_GAS_VALVE )
   END_RUNG
   RUNG wire#w1
      Move(in := 0.0, out1 => #ACTIONS_SEQUENCE.SETPOINT_PRESSURE)
      wire#w2
      R_Coil( #ACTIONS_SEQUENCE.REQ_STOP_PRESSURE_GAS_CONTROL )
   END_RUNG
   RUNG wire#w2
      R_Coil( #ACTIONS_SEQUENCE.REQ_START_PRESSURE_GAS_CONTROL )
   END_RUNG
   RUNG wire#w1
      Move(in := 0, out1 => #ACTIONS_SEQUENCE.SETPOINT_MOTOR_STIRRER)
      wire#w3
      R_Coil( #ACTIONS_SEQUENCE.REQUEST_STOP_MOTOR_STIRRER )
   END_RUNG
   RUNG wire#w3
      R_Coil( #ACTIONS_SEQUENCE.REQUEST_START_MOTOR_STIRRER )
   END_RUNG
   RUNG wire#w1
      R_Coil( #ACTIONS_SEQUENCE.REQ_STOP_TRANSFER_POWDER_VALVE )
   END_RUNG
   RUNG wire#w1
      R_Coil( #ACTIONS_SEQUENCE.REQ_START_TRANSFER_POWDER_VALVE )
   END_RUNG
   RUNG wire#w1
      R_Coil( #CONTROL_SEQUENCE.MATERIAL_APPLIED )
   END_RUNG
   // the same network as SCL:
   IF #DATA_SEQUENCE.STEP_9 THEN
       #ACTIONS_SEQUENCE.REQ_STOP_PRESSURE_GAS_VALVE := FALSE;
       #ACTIONS_SEQUENCE.REQ_STOP_PRESSURE_GAS_VALVE := FALSE;
       #ACTIONS_SEQUENCE.REQ_STOP_RELIEF_GAS_VALVE := TRUE;
       #ACTIONS_SEQUENCE.REQ_START_RELIEF_GAS_VALVE := FALSE;
       #ACTIONS_SEQUENCE.SETPOINT_PRESSURE := 0.0;
       #ACTIONS_SEQUENCE.REQ_STOP_PRESSURE_GAS_CONTROL := FALSE;
       #ACTIONS_SEQUENCE.REQ_START_PRESSURE_GAS_CONTROL := FALSE;
       #ACTIONS_SEQUENCE.SETPOINT_MOTOR_STIRRER := 0;
       #ACTIONS_SEQUENCE.REQUEST_STOP_MOTOR_STIRRER := FALSE;
       #ACTIONS_SEQUENCE.REQUEST_START_MOTOR_STIRRER := FALSE;
       #ACTIONS_SEQUENCE.REQ_STOP_TRANSFER_POWDER_VALVE := FALSE;
       #ACTIONS_SEQUENCE.REQ_START_TRANSFER_POWDER_VALVE := FALSE;
       #CONTROL_SEQUENCE.MATERIAL_APPLIED := FALSE;
   END_IF;
END_REGION

REGION Network 30: STEP 1 TO STEP 2
   RUNG wire#powerrail
      Contact( #DATA_SEQUENCE.SEQUENCE_RUNNING )
      wire#w1
      Contact( #DATA_SEQUENCE.STEP_1 )
      Contact( #CONTROL_SEQUENCE.HOPPER_PRESSURE_IN_RANGE )
      Contact( #CONTROL_SEQUENCE.HOPPER_MOTOR_STIRRER_IN_RANGE )
      wire#w2
      I_Contact( #DATA_SEQUENCE.STEP_3 )
      I_Contact( #DATA_SEQUENCE.STEP_4 )
      I_Contact( #DATA_SEQUENCE.STEP_5 )
      I_Contact( #DATA_SEQUENCE.STEP_6 )
      I_Contact( #DATA_SEQUENCE.STEP_7 )
      I_Contact( #DATA_SEQUENCE.STEP_8 )
      Coil( #DATA_SEQUENCE.STEP_2 )
   END_RUNG
   RUNG wire#w1
      Contact( #DATA_SEQUENCE.STEP_2 )
   END_RUNG wire#w2
   // the same network as SCL:
   #DATA_SEQUENCE.STEP_2 := #DATA_SEQUENCE.SEQUENCE_RUNNING AND ((#DATA_SEQUENCE.STEP_1 AND #CONTROL_SEQUENCE.HOPPER_PRESSURE_IN_RANGE AND #CONTROL_SEQUENCE.HOPPER_MOTOR_STIRRER_IN_RANGE) OR #DATA_SEQUENCE.STEP_2) AND NOT #DATA_SEQUENCE.STEP_3 AND NOT #DATA_SEQUENCE.STEP_4 AND NOT #DATA_SEQUENCE.STEP_5 AND NOT #DATA_SEQUENCE.STEP_6 AND NOT #DATA_SEQUENCE.STEP_7 AND NOT #DATA_SEQUENCE.STEP_8;
END_REGION

REGION Network 31: STEP 2, 6, 4 TO STEP 3
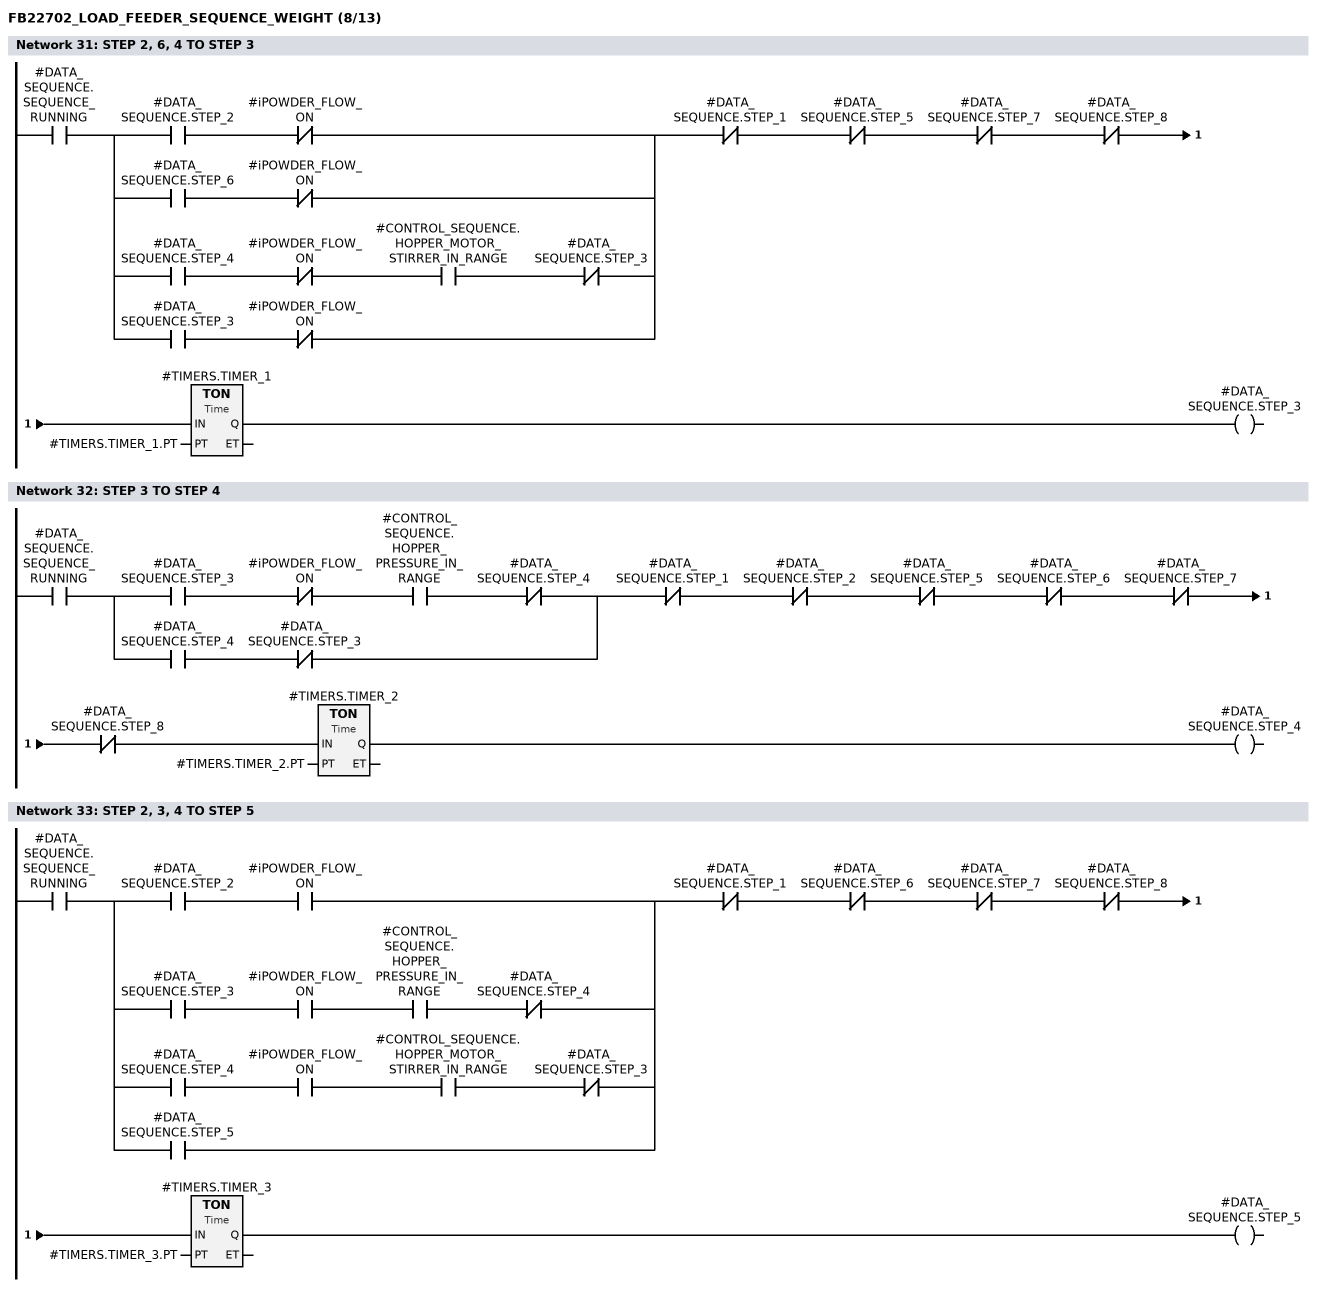
   RUNG wire#powerrail
      Contact( #DATA_SEQUENCE.SEQUENCE_RUNNING )
      wire#w1
      Contact( #DATA_SEQUENCE.STEP_2 )
      I_Contact( #iPOWDER_FLOW_ON )
      wire#w2
      I_Contact( #DATA_SEQUENCE.STEP_1 )
      I_Contact( #DATA_SEQUENCE.STEP_5 )
      I_Contact( #DATA_SEQUENCE.STEP_7 )
      I_Contact( #DATA_SEQUENCE.STEP_8 )
      { S7_Templates := "time_type := Time" } #TIMERS.TIMER_1.TON(pt := #TIMERS.TIMER_1.PT, et =>)
      Coil( #DATA_SEQUENCE.STEP_3 )
   END_RUNG
   RUNG wire#w1
      Contact( #DATA_SEQUENCE.STEP_6 )
      I_Contact( #iPOWDER_FLOW_ON )
   END_RUNG wire#w2
   RUNG wire#w1
      Contact( #DATA_SEQUENCE.STEP_4 )
      I_Contact( #iPOWDER_FLOW_ON )
      Contact( #CONTROL_SEQUENCE.HOPPER_MOTOR_STIRRER_IN_RANGE )
      I_Contact( #DATA_SEQUENCE.STEP_3 )
   END_RUNG wire#w2
   RUNG wire#w1
      Contact( #DATA_SEQUENCE.STEP_3 )
      I_Contact( #iPOWDER_FLOW_ON )
   END_RUNG wire#w2
   // the same network as SCL:
   #TIMERS.TIMER_1.TON(IN := #DATA_SEQUENCE.SEQUENCE_RUNNING AND ((#DATA_SEQUENCE.STEP_2 AND NOT #iPOWDER_FLOW_ON) OR (#DATA_SEQUENCE.STEP_6 AND NOT #iPOWDER_FLOW_ON) OR (#DATA_SEQUENCE.STEP_4 AND NOT #iPOWDER_FLOW_ON AND #CONTROL_SEQUENCE.HOPPER_MOTOR_STIRRER_IN_RANGE AND NOT #DATA_SEQUENCE.STEP_3) OR (#DATA_SEQUENCE.STEP_3 AND NOT #iPOWDER_FLOW_ON)) AND NOT #DATA_SEQUENCE.STEP_1 AND NOT #DATA_SEQUENCE.STEP_5 AND NOT #DATA_SEQUENCE.STEP_7 AND NOT #DATA_SEQUENCE.STEP_8,
                       PT := #TIMERS.TIMER_1.PT);
   #DATA_SEQUENCE.STEP_3 := #TIMERS.TIMER_1.Q;
END_REGION

REGION Network 32: STEP 3 TO STEP 4
   RUNG wire#powerrail
      Contact( #DATA_SEQUENCE.SEQUENCE_RUNNING )
      wire#w1
      Contact( #DATA_SEQUENCE.STEP_3 )
      I_Contact( #iPOWDER_FLOW_ON )
      Contact( #CONTROL_SEQUENCE.HOPPER_PRESSURE_IN_RANGE )
      I_Contact( #DATA_SEQUENCE.STEP_4 )
      wire#w2
      I_Contact( #DATA_SEQUENCE.STEP_1 )
      I_Contact( #DATA_SEQUENCE.STEP_2 )
      I_Contact( #DATA_SEQUENCE.STEP_5 )
      I_Contact( #DATA_SEQUENCE.STEP_6 )
      I_Contact( #DATA_SEQUENCE.STEP_7 )
      I_Contact( #DATA_SEQUENCE.STEP_8 )
      { S7_Templates := "time_type := Time" } #TIMERS.TIMER_2.TON(pt := #TIMERS.TIMER_2.PT, et =>)
      Coil( #DATA_SEQUENCE.STEP_4 )
   END_RUNG
   RUNG wire#w1
      Contact( #DATA_SEQUENCE.STEP_4 )
      I_Contact( #DATA_SEQUENCE.STEP_3 )
   END_RUNG wire#w2
   // the same network as SCL:
   #TIMERS.TIMER_2.TON(IN := #DATA_SEQUENCE.SEQUENCE_RUNNING AND ((#DATA_SEQUENCE.STEP_3 AND NOT #iPOWDER_FLOW_ON AND #CONTROL_SEQUENCE.HOPPER_PRESSURE_IN_RANGE AND NOT #DATA_SEQUENCE.STEP_4) OR (#DATA_SEQUENCE.STEP_4 AND NOT #DATA_SEQUENCE.STEP_3)) AND NOT #DATA_SEQUENCE.STEP_1 AND NOT #DATA_SEQUENCE.STEP_2 AND NOT #DATA_SEQUENCE.STEP_5 AND NOT #DATA_SEQUENCE.STEP_6 AND NOT #DATA_SEQUENCE.STEP_7 AND NOT #DATA_SEQUENCE.STEP_8,
                       PT := #TIMERS.TIMER_2.PT);
   #DATA_SEQUENCE.STEP_4 := #TIMERS.TIMER_2.Q;
END_REGION

REGION Network 33: STEP 2, 3, 4 TO STEP 5
   RUNG wire#powerrail
      Contact( #DATA_SEQUENCE.SEQUENCE_RUNNING )
      wire#w1
      Contact( #DATA_SEQUENCE.STEP_2 )
      Contact( #iPOWDER_FLOW_ON )
      wire#w2
      I_Contact( #DATA_SEQUENCE.STEP_1 )
      I_Contact( #DATA_SEQUENCE.STEP_6 )
      I_Contact( #DATA_SEQUENCE.STEP_7 )
      I_Contact( #DATA_SEQUENCE.STEP_8 )
      { S7_Templates := "time_type := Time" } #TIMERS.TIMER_3.TON(pt := #TIMERS.TIMER_3.PT, et =>)
      Coil( #DATA_SEQUENCE.STEP_5 )
   END_RUNG
   RUNG wire#w1
      Contact( #DATA_SEQUENCE.STEP_3 )
      Contact( #iPOWDER_FLOW_ON )
      Contact( #CONTROL_SEQUENCE.HOPPER_PRESSURE_IN_RANGE )
      I_Contact( #DATA_SEQUENCE.STEP_4 )
   END_RUNG wire#w2
   RUNG wire#w1
      Contact( #DATA_SEQUENCE.STEP_4 )
      Contact( #iPOWDER_FLOW_ON )
      Contact( #CONTROL_SEQUENCE.HOPPER_MOTOR_STIRRER_IN_RANGE )
      I_Contact( #DATA_SEQUENCE.STEP_3 )
   END_RUNG wire#w2
   RUNG wire#w1
      Contact( #DATA_SEQUENCE.STEP_5 )
   END_RUNG wire#w2
   // the same network as SCL:
   #TIMERS.TIMER_3.TON(IN := #DATA_SEQUENCE.SEQUENCE_RUNNING AND ((#DATA_SEQUENCE.STEP_2 AND #iPOWDER_FLOW_ON) OR (#DATA_SEQUENCE.STEP_3 AND #iPOWDER_FLOW_ON AND #CONTROL_SEQUENCE.HOPPER_PRESSURE_IN_RANGE AND NOT #DATA_SEQUENCE.STEP_4) OR (#DATA_SEQUENCE.STEP_4 AND #iPOWDER_FLOW_ON AND #CONTROL_SEQUENCE.HOPPER_MOTOR_STIRRER_IN_RANGE AND NOT #DATA_SEQUENCE.STEP_3) OR #DATA_SEQUENCE.STEP_5) AND NOT #DATA_SEQUENCE.STEP_1 AND NOT #DATA_SEQUENCE.STEP_6 AND NOT #DATA_SEQUENCE.STEP_7 AND NOT #DATA_SEQUENCE.STEP_8,
                       PT := #TIMERS.TIMER_3.PT);
   #DATA_SEQUENCE.STEP_5 := #TIMERS.TIMER_3.Q;
END_REGION

REGION Network 34: STEP 5 AND STOP COMMAND TO STEP 7
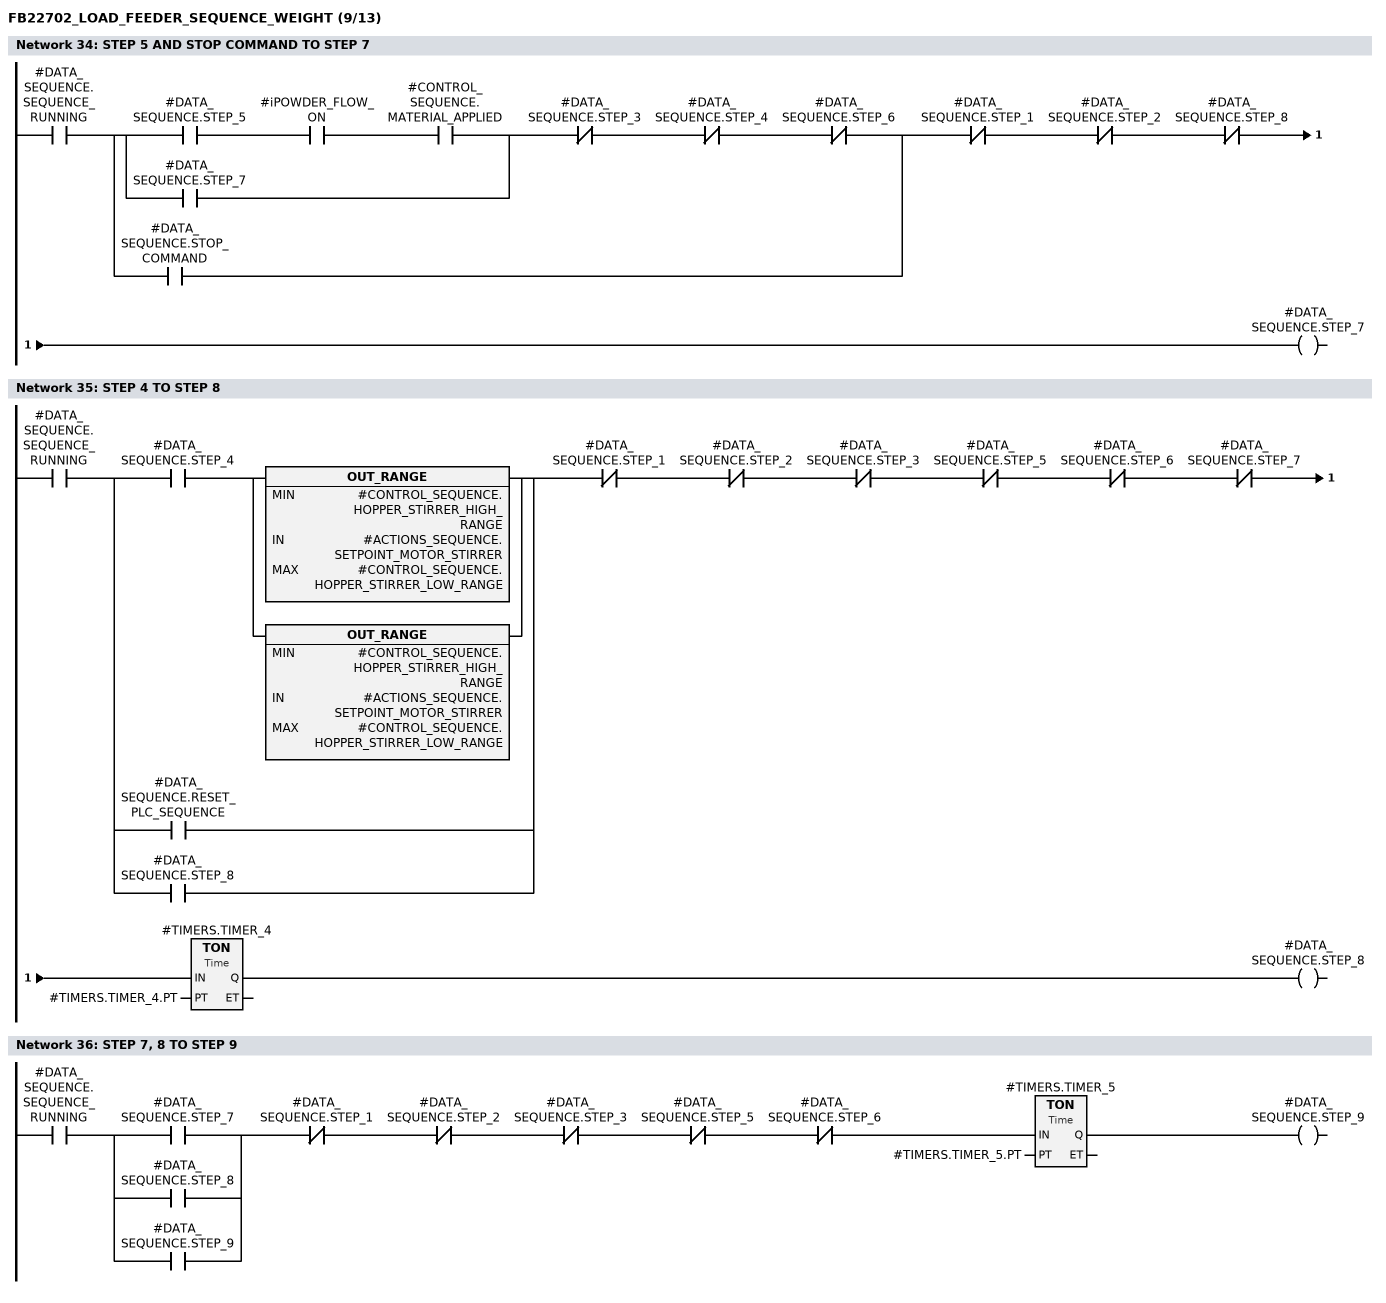
   RUNG wire#powerrail
      Contact( #DATA_SEQUENCE.SEQUENCE_RUNNING )
      wire#w1
      Contact( #DATA_SEQUENCE.STEP_5 )
      Contact( #iPOWDER_FLOW_ON )
      Contact( #CONTROL_SEQUENCE.MATERIAL_APPLIED )
      wire#w2
      I_Contact( #DATA_SEQUENCE.STEP_3 )
      I_Contact( #DATA_SEQUENCE.STEP_4 )
      I_Contact( #DATA_SEQUENCE.STEP_6 )
      wire#w3
      I_Contact( #DATA_SEQUENCE.STEP_1 )
      I_Contact( #DATA_SEQUENCE.STEP_2 )
      I_Contact( #DATA_SEQUENCE.STEP_8 )
      Coil( #DATA_SEQUENCE.STEP_7 )
   END_RUNG
   RUNG wire#w1
      Contact( #DATA_SEQUENCE.STEP_7 )
   END_RUNG wire#w2
   RUNG wire#w1
      Contact( #DATA_SEQUENCE.STOP_COMMAND )
   END_RUNG wire#w3
   // the same network as SCL:
   #DATA_SEQUENCE.STEP_7 := #DATA_SEQUENCE.SEQUENCE_RUNNING AND ((((#DATA_SEQUENCE.STEP_5 AND #iPOWDER_FLOW_ON AND #CONTROL_SEQUENCE.MATERIAL_APPLIED) OR #DATA_SEQUENCE.STEP_7) AND NOT #DATA_SEQUENCE.STEP_3 AND NOT #DATA_SEQUENCE.STEP_4 AND NOT #DATA_SEQUENCE.STEP_6) OR #DATA_SEQUENCE.STOP_COMMAND) AND NOT #DATA_SEQUENCE.STEP_1 AND NOT #DATA_SEQUENCE.STEP_2 AND NOT #DATA_SEQUENCE.STEP_8;
END_REGION

REGION Network 35: STEP 4 TO STEP 8
   #TIMERS.TIMER_4.TON(IN := #DATA_SEQUENCE.SEQUENCE_RUNNING AND ((#DATA_SEQUENCE.STEP_4 AND ((#ACTIONS_SEQUENCE.SETPOINT_MOTOR_STIRRER < #CONTROL_SEQUENCE.HOPPER_STIRRER_HIGH_RANGE) OR (#ACTIONS_SEQUENCE.SETPOINT_MOTOR_STIRRER > #CONTROL_SEQUENCE.HOPPER_STIRRER_LOW_RANGE) OR (#ACTIONS_SEQUENCE.SETPOINT_MOTOR_STIRRER < #CONTROL_SEQUENCE.HOPPER_STIRRER_HIGH_RANGE) OR (#ACTIONS_SEQUENCE.SETPOINT_MOTOR_STIRRER > #CONTROL_SEQUENCE.HOPPER_STIRRER_LOW_RANGE))) OR #DATA_SEQUENCE.RESET_PLC_SEQUENCE OR #DATA_SEQUENCE.STEP_8) AND NOT #DATA_SEQUENCE.STEP_1 AND NOT #DATA_SEQUENCE.STEP_2 AND NOT #DATA_SEQUENCE.STEP_3 AND NOT #DATA_SEQUENCE.STEP_5 AND NOT #DATA_SEQUENCE.STEP_6 AND NOT #DATA_SEQUENCE.STEP_7,
                       PT := #TIMERS.TIMER_4.PT);
   #DATA_SEQUENCE.STEP_8 := #TIMERS.TIMER_4.Q;
END_REGION

REGION Network 36: STEP 7, 8 TO STEP 9
   RUNG wire#powerrail
      Contact( #DATA_SEQUENCE.SEQUENCE_RUNNING )
      wire#w1
      Contact( #DATA_SEQUENCE.STEP_7 )
      wire#w2
      I_Contact( #DATA_SEQUENCE.STEP_1 )
      I_Contact( #DATA_SEQUENCE.STEP_2 )
      I_Contact( #DATA_SEQUENCE.STEP_3 )
      I_Contact( #DATA_SEQUENCE.STEP_5 )
      I_Contact( #DATA_SEQUENCE.STEP_6 )
      { S7_Templates := "time_type := Time" } #TIMERS.TIMER_5.TON(pt := #TIMERS.TIMER_5.PT, et =>)
      Coil( #DATA_SEQUENCE.STEP_9 )
   END_RUNG
   RUNG wire#w1
      Contact( #DATA_SEQUENCE.STEP_8 )
   END_RUNG wire#w2
   RUNG wire#w1
      Contact( #DATA_SEQUENCE.STEP_9 )
   END_RUNG wire#w2
   // the same network as SCL:
   #TIMERS.TIMER_5.TON(IN := #DATA_SEQUENCE.SEQUENCE_RUNNING AND (#DATA_SEQUENCE.STEP_7 OR #DATA_SEQUENCE.STEP_8 OR #DATA_SEQUENCE.STEP_9) AND NOT #DATA_SEQUENCE.STEP_1 AND NOT #DATA_SEQUENCE.STEP_2 AND NOT #DATA_SEQUENCE.STEP_3 AND NOT #DATA_SEQUENCE.STEP_5 AND NOT #DATA_SEQUENCE.STEP_6,
                       PT := #TIMERS.TIMER_5.PT);
   #DATA_SEQUENCE.STEP_9 := #TIMERS.TIMER_5.Q;
END_REGION

REGION Network 37: STEP 9 TO SEQUENCE DONE
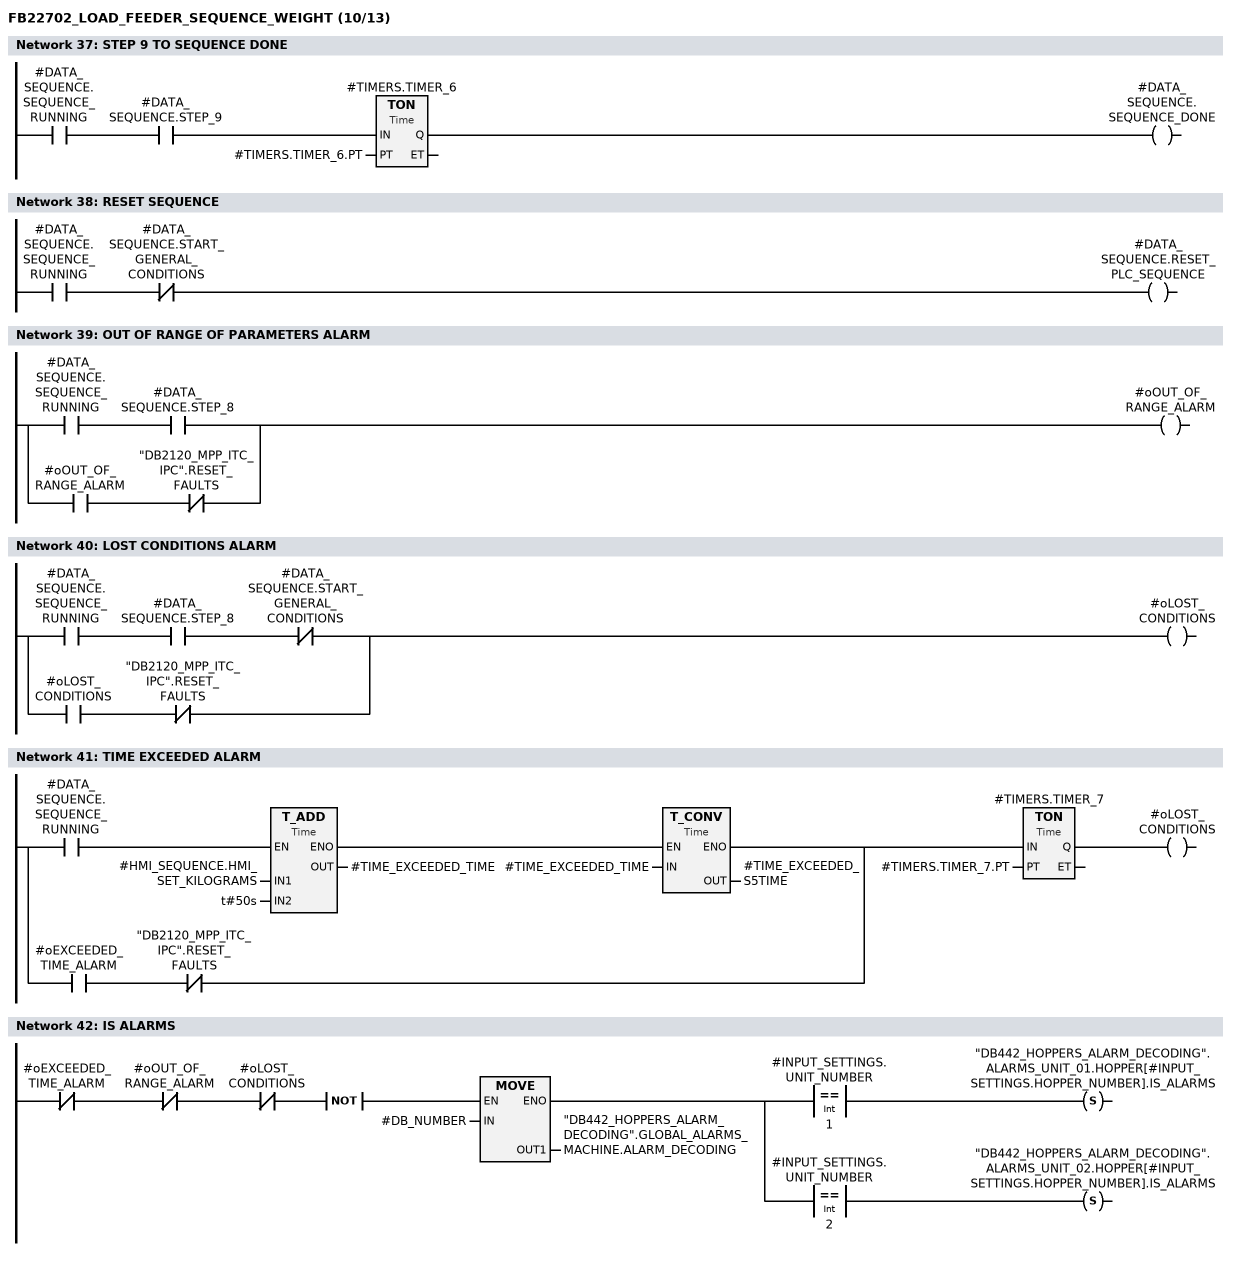
   RUNG wire#powerrail
      Contact( #DATA_SEQUENCE.SEQUENCE_RUNNING )
      Contact( #DATA_SEQUENCE.STEP_9 )
      { S7_Templates := "time_type := Time" } #TIMERS.TIMER_6.TON(pt := #TIMERS.TIMER_6.PT, et =>)
      Coil( #DATA_SEQUENCE.SEQUENCE_DONE )
   END_RUNG
   // the same network as SCL:
   #TIMERS.TIMER_6.TON(IN := #DATA_SEQUENCE.SEQUENCE_RUNNING AND #DATA_SEQUENCE.STEP_9,
                       PT := #TIMERS.TIMER_6.PT);
   #DATA_SEQUENCE.SEQUENCE_DONE := #TIMERS.TIMER_6.Q;
END_REGION

REGION Network 38: RESET SEQUENCE
   RUNG wire#powerrail
      Contact( #DATA_SEQUENCE.SEQUENCE_RUNNING )
      I_Contact( #DATA_SEQUENCE.START_GENERAL_CONDITIONS )
      Coil( #DATA_SEQUENCE.RESET_PLC_SEQUENCE )
   END_RUNG
   // the same network as SCL:
   #DATA_SEQUENCE.RESET_PLC_SEQUENCE := #DATA_SEQUENCE.SEQUENCE_RUNNING AND NOT #DATA_SEQUENCE.START_GENERAL_CONDITIONS;
END_REGION

REGION Network 39: OUT OF RANGE OF PARAMETERS ALARM
   RUNG wire#powerrail
      Contact( #DATA_SEQUENCE.SEQUENCE_RUNNING )
      Contact( #DATA_SEQUENCE.STEP_8 )
      wire#w1
      Coil( #oOUT_OF_RANGE_ALARM )
   END_RUNG
   RUNG wire#powerrail
      Contact( #oOUT_OF_RANGE_ALARM )
      I_Contact( "DB2120_MPP_ITC_IPC".RESET_FAULTS )
   END_RUNG wire#w1
   // the same network as SCL:
   #oOUT_OF_RANGE_ALARM := (#DATA_SEQUENCE.SEQUENCE_RUNNING AND #DATA_SEQUENCE.STEP_8) OR (#oOUT_OF_RANGE_ALARM AND NOT "DB2120_MPP_ITC_IPC".RESET_FAULTS);
END_REGION

REGION Network 40: LOST CONDITIONS ALARM
   RUNG wire#powerrail
      Contact( #DATA_SEQUENCE.SEQUENCE_RUNNING )
      Contact( #DATA_SEQUENCE.STEP_8 )
      I_Contact( #DATA_SEQUENCE.START_GENERAL_CONDITIONS )
      wire#w1
      Coil( #oLOST_CONDITIONS )
   END_RUNG
   RUNG wire#powerrail
      Contact( #oLOST_CONDITIONS )
      I_Contact( "DB2120_MPP_ITC_IPC".RESET_FAULTS )
   END_RUNG wire#w1
   // the same network as SCL:
   #oLOST_CONDITIONS := (#DATA_SEQUENCE.SEQUENCE_RUNNING AND #DATA_SEQUENCE.STEP_8 AND NOT #DATA_SEQUENCE.START_GENERAL_CONDITIONS) OR (#oLOST_CONDITIONS AND NOT "DB2120_MPP_ITC_IPC".RESET_FAULTS);
END_REGION

REGION Network 41: TIME EXCEEDED ALARM
   RUNG wire#powerrail
      Contact( #DATA_SEQUENCE.SEQUENCE_RUNNING )
      { S7_Templates := "[date_type := Time, time_type := Time]" } T_ADD(IN1 := #HMI_SEQUENCE.HMI_SET_KILOGRAMS, IN2 := t#50s, OUT => #TIME_EXCEEDED_TIME)
      { S7_Templates := "[src_type := Time, dest_type := S5Time]" } T_CONV(IN := #TIME_EXCEEDED_TIME, OUT => #TIME_EXCEEDED_S5TIME)
      wire#w1
      { S7_Templates := "time_type := Time" } #TIMERS.TIMER_7.TON(pt := #TIMERS.TIMER_7.PT, et =>)
      Coil( #oLOST_CONDITIONS )
   END_RUNG
   RUNG wire#powerrail
      Contact( #oEXCEEDED_TIME_ALARM )
      I_Contact( "DB2120_MPP_ITC_IPC".RESET_FAULTS )
   END_RUNG wire#w1
   // the same network as SCL:
   T_ADD(EN := #DATA_SEQUENCE.SEQUENCE_RUNNING,
         IN1 := #HMI_SEQUENCE.HMI_SET_KILOGRAMS,
         IN2 := t#50s,
         OUT => #TIME_EXCEEDED_TIME,
         ENO => #_w1);
   T_CONV(EN := #_w1, IN := #TIME_EXCEEDED_TIME, OUT => #TIME_EXCEEDED_S5TIME, ENO => #_w2);
   #TIMERS.TIMER_7.TON(IN := #_w2 OR (#oEXCEEDED_TIME_ALARM AND NOT "DB2120_MPP_ITC_IPC".RESET_FAULTS),
                       PT := #TIMERS.TIMER_7.PT);
   #oLOST_CONDITIONS := #TIMERS.TIMER_7.Q;
END_REGION

REGION Network 42: IS ALARMS
   RUNG wire#powerrail
      I_Contact( #oEXCEEDED_TIME_ALARM )
      I_Contact( #oOUT_OF_RANGE_ALARM )
      I_Contact( #oLOST_CONDITIONS )
      Not()
      { S7_GenerateENO := "TRUE" } Move(in := #DB_NUMBER, out1 => "DB442_HOPPERS_ALARM_DECODING".GLOBAL_ALARMS_MACHINE.ALARM_DECODING)
      wire#w1
      { S7_Templates := "SrcType := Int" } EQ_Contact(in1 := #INPUT_SETTINGS.UNIT_NUMBER, in2 := 1)
      S_Coil( "DB442_HOPPERS_ALARM_DECODING".ALARMS_UNIT_01.HOPPER[#INPUT_SETTINGS.HOPPER_NUMBER].IS_ALARMS )
   END_RUNG
   RUNG wire#w1
      { S7_Templates := "SrcType := Int" } EQ_Contact(in1 := #INPUT_SETTINGS.UNIT_NUMBER, in2 := 2)
      S_Coil( "DB442_HOPPERS_ALARM_DECODING".ALARMS_UNIT_02.HOPPER[#INPUT_SETTINGS.HOPPER_NUMBER].IS_ALARMS )
   END_RUNG
   // the same network as SCL:
   // ENO of a box is taken as its EN; it also drops when the box reports an error
   #_w1 := NOT (NOT #oEXCEEDED_TIME_ALARM AND NOT #oOUT_OF_RANGE_ALARM AND NOT #oLOST_CONDITIONS);
   IF #_w1 THEN "DB442_HOPPERS_ALARM_DECODING".GLOBAL_ALARMS_MACHINE.ALARM_DECODING := #DB_NUMBER; END_IF;
   IF #_w1 AND (#INPUT_SETTINGS.UNIT_NUMBER = 1) THEN
       "DB442_HOPPERS_ALARM_DECODING".ALARMS_UNIT_01.HOPPER[#INPUT_SETTINGS.HOPPER_NUMBER].IS_ALARMS := TRUE;
   END_IF;
   IF #_w1 AND (#INPUT_SETTINGS.UNIT_NUMBER = 2) THEN
       "DB442_HOPPERS_ALARM_DECODING".ALARMS_UNIT_02.HOPPER[#INPUT_SETTINGS.HOPPER_NUMBER].IS_ALARMS := TRUE;
   END_IF;
END_REGION

REGION Network 43: MANUAL START HELP / General Conditions Help
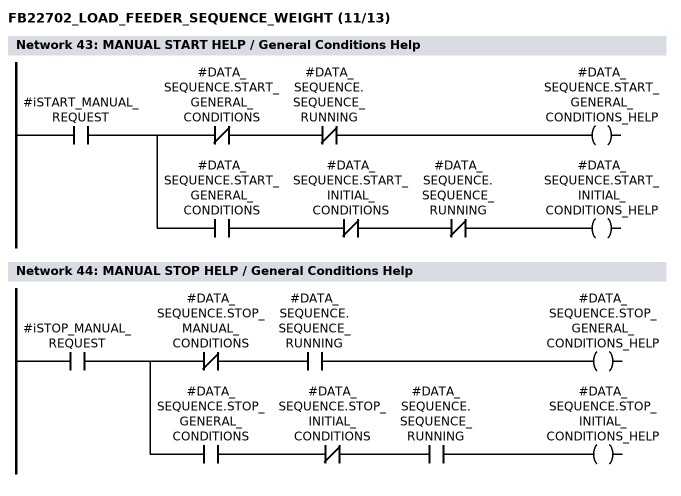
   RUNG wire#powerrail
      Contact( #iSTART_MANUAL_REQUEST )
      wire#w1
      I_Contact( #DATA_SEQUENCE.START_GENERAL_CONDITIONS )
      I_Contact( #DATA_SEQUENCE.SEQUENCE_RUNNING )
      Coil( #DATA_SEQUENCE.START_GENERAL_CONDITIONS_HELP )
   END_RUNG
   RUNG wire#w1
      Contact( #DATA_SEQUENCE.START_GENERAL_CONDITIONS )
      I_Contact( #DATA_SEQUENCE.START_INITIAL_CONDITIONS )
      I_Contact( #DATA_SEQUENCE.SEQUENCE_RUNNING )
      Coil( #DATA_SEQUENCE.START_INITIAL_CONDITIONS_HELP )
   END_RUNG
   // the same network as SCL:
   #DATA_SEQUENCE.START_GENERAL_CONDITIONS_HELP := #iSTART_MANUAL_REQUEST AND NOT #DATA_SEQUENCE.START_GENERAL_CONDITIONS AND NOT #DATA_SEQUENCE.SEQUENCE_RUNNING;
   #DATA_SEQUENCE.START_INITIAL_CONDITIONS_HELP := #iSTART_MANUAL_REQUEST AND #DATA_SEQUENCE.START_GENERAL_CONDITIONS AND NOT #DATA_SEQUENCE.START_INITIAL_CONDITIONS AND NOT #DATA_SEQUENCE.SEQUENCE_RUNNING;
END_REGION

REGION Network 44: MANUAL STOP HELP / General Conditions Help
   RUNG wire#powerrail
      Contact( #iSTOP_MANUAL_REQUEST )
      wire#w1
      I_Contact( #DATA_SEQUENCE.STOP_MANUAL_CONDITIONS )
      Contact( #DATA_SEQUENCE.SEQUENCE_RUNNING )
      Coil( #DATA_SEQUENCE.STOP_GENERAL_CONDITIONS_HELP )
   END_RUNG
   RUNG wire#w1
      Contact( #DATA_SEQUENCE.STOP_GENERAL_CONDITIONS )
      I_Contact( #DATA_SEQUENCE.STOP_INITIAL_CONDITIONS )
      Contact( #DATA_SEQUENCE.SEQUENCE_RUNNING )
      Coil( #DATA_SEQUENCE.STOP_INITIAL_CONDITIONS_HELP )
   END_RUNG
   // the same network as SCL:
   #DATA_SEQUENCE.STOP_GENERAL_CONDITIONS_HELP := #iSTOP_MANUAL_REQUEST AND NOT #DATA_SEQUENCE.STOP_MANUAL_CONDITIONS AND #DATA_SEQUENCE.SEQUENCE_RUNNING;
   #DATA_SEQUENCE.STOP_INITIAL_CONDITIONS_HELP := #iSTOP_MANUAL_REQUEST AND #DATA_SEQUENCE.STOP_GENERAL_CONDITIONS AND NOT #DATA_SEQUENCE.STOP_INITIAL_CONDITIONS AND #DATA_SEQUENCE.SEQUENCE_RUNNING;
END_REGION

REGION Network 45: HMI SEQUENCE STATUS
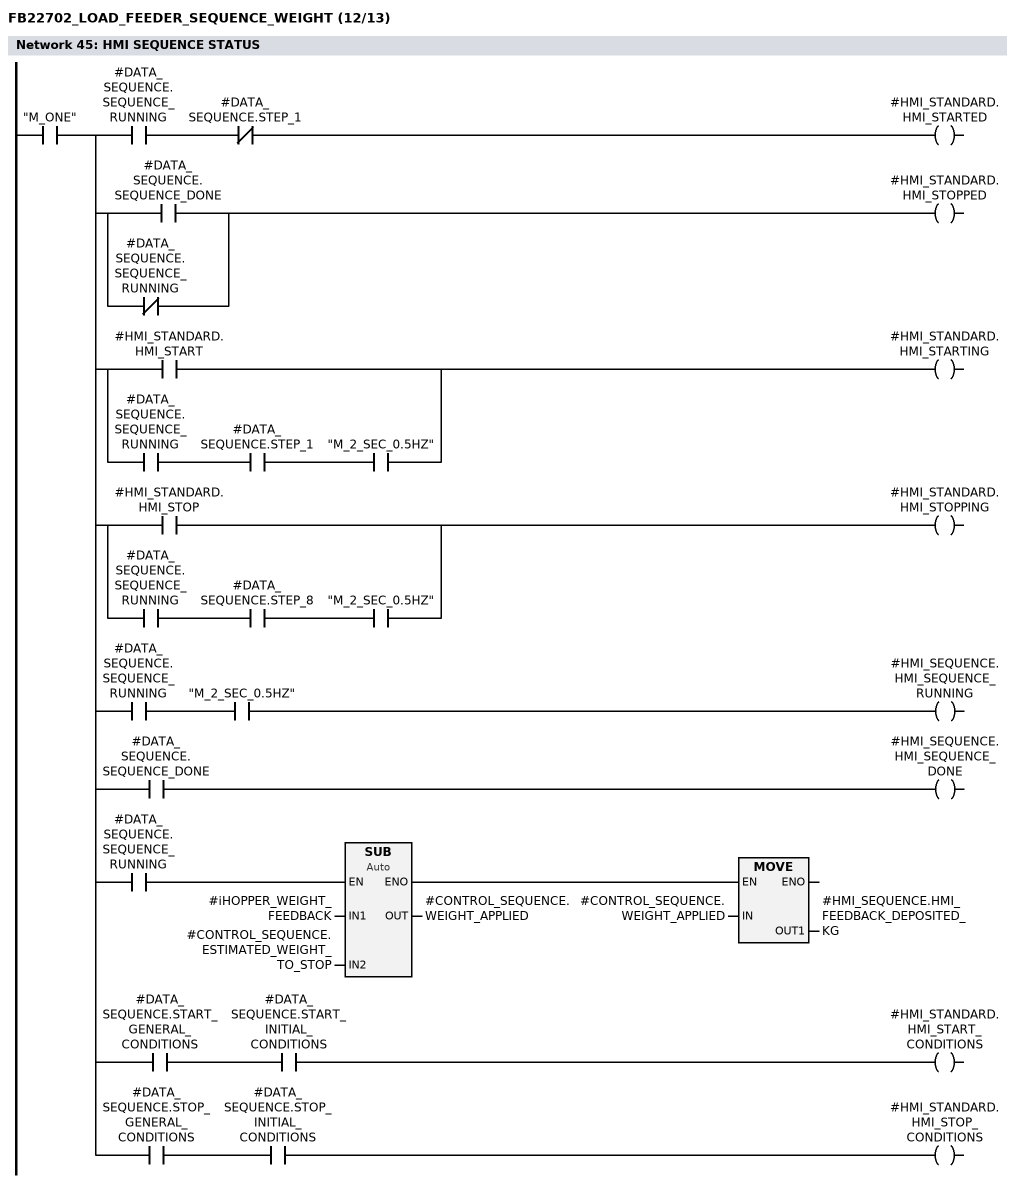
   RUNG wire#powerrail
      Contact( "M_ONE" )
      wire#w1
      Contact( #DATA_SEQUENCE.SEQUENCE_RUNNING )
      I_Contact( #DATA_SEQUENCE.STEP_1 )
      Coil( #HMI_STANDARD.HMI_STARTED )
   END_RUNG
   RUNG wire#w1
      Contact( #DATA_SEQUENCE.SEQUENCE_DONE )
      wire#w2
      Coil( #HMI_STANDARD.HMI_STOPPED )
   END_RUNG
   RUNG wire#w1
      I_Contact( #DATA_SEQUENCE.SEQUENCE_RUNNING )
   END_RUNG wire#w2
   RUNG wire#w1
      Contact( #HMI_STANDARD.HMI_START )
      wire#w3
      Coil( #HMI_STANDARD.HMI_STARTING )
   END_RUNG
   RUNG wire#w1
      Contact( #DATA_SEQUENCE.SEQUENCE_RUNNING )
      Contact( #DATA_SEQUENCE.STEP_1 )
      Contact( "M_2_SEC_0.5HZ" )
   END_RUNG wire#w3
   RUNG wire#w1
      Contact( #HMI_STANDARD.HMI_STOP )
      wire#w4
      Coil( #HMI_STANDARD.HMI_STOPPING )
   END_RUNG
   RUNG wire#w1
      Contact( #DATA_SEQUENCE.SEQUENCE_RUNNING )
      Contact( #DATA_SEQUENCE.STEP_8 )
      Contact( "M_2_SEC_0.5HZ" )
   END_RUNG wire#w4
   RUNG wire#w1
      Contact( #DATA_SEQUENCE.SEQUENCE_RUNNING )
      Contact( "M_2_SEC_0.5HZ" )
      Coil( #HMI_SEQUENCE.HMI_SEQUENCE_RUNNING )
   END_RUNG
   RUNG wire#w1
      Contact( #DATA_SEQUENCE.SEQUENCE_DONE )
      Coil( #HMI_SEQUENCE.HMI_SEQUENCE_DONE )
   END_RUNG
   RUNG wire#w1
      Contact( #DATA_SEQUENCE.SEQUENCE_RUNNING )
      Sub(in1 := #iHOPPER_WEIGHT_FEEDBACK, in2 := #CONTROL_SEQUENCE.ESTIMATED_WEIGHT_TO_STOP, out => #CONTROL_SEQUENCE.WEIGHT_APPLIED)
      Move(in := #CONTROL_SEQUENCE.WEIGHT_APPLIED, out1 => #HMI_SEQUENCE.HMI_FEEDBACK_DEPOSITED_KG)
   END_RUNG
   RUNG wire#w1
      Contact( #DATA_SEQUENCE.START_GENERAL_CONDITIONS )
      Contact( #DATA_SEQUENCE.START_INITIAL_CONDITIONS )
      Coil( #HMI_STANDARD.HMI_START_CONDITIONS )
   END_RUNG
   RUNG wire#w1
      Contact( #DATA_SEQUENCE.STOP_GENERAL_CONDITIONS )
      Contact( #DATA_SEQUENCE.STOP_INITIAL_CONDITIONS )
      Coil( #HMI_STANDARD.HMI_STOP_CONDITIONS )
   END_RUNG
   // the same network as SCL:
   #HMI_STANDARD.HMI_STARTED := "M_ONE" AND #DATA_SEQUENCE.SEQUENCE_RUNNING AND NOT #DATA_SEQUENCE.STEP_1;
   #HMI_STANDARD.HMI_STOPPED := "M_ONE" AND (#DATA_SEQUENCE.SEQUENCE_DONE OR NOT #DATA_SEQUENCE.SEQUENCE_RUNNING);
   #HMI_STANDARD.HMI_STARTING := "M_ONE" AND (#HMI_STANDARD.HMI_START OR (#DATA_SEQUENCE.SEQUENCE_RUNNING AND #DATA_SEQUENCE.STEP_1 AND "M_2_SEC_0.5HZ"));
   #HMI_STANDARD.HMI_STOPPING := "M_ONE" AND (#HMI_STANDARD.HMI_STOP OR (#DATA_SEQUENCE.SEQUENCE_RUNNING AND #DATA_SEQUENCE.STEP_8 AND "M_2_SEC_0.5HZ"));
   #HMI_SEQUENCE.HMI_SEQUENCE_RUNNING := "M_ONE" AND #DATA_SEQUENCE.SEQUENCE_RUNNING AND "M_2_SEC_0.5HZ";
   #HMI_SEQUENCE.HMI_SEQUENCE_DONE := "M_ONE" AND #DATA_SEQUENCE.SEQUENCE_DONE;
   IF "M_ONE" AND #DATA_SEQUENCE.SEQUENCE_RUNNING THEN
       #CONTROL_SEQUENCE.WEIGHT_APPLIED := #iHOPPER_WEIGHT_FEEDBACK - #CONTROL_SEQUENCE.ESTIMATED_WEIGHT_TO_STOP;
       #HMI_SEQUENCE.HMI_FEEDBACK_DEPOSITED_KG := #CONTROL_SEQUENCE.WEIGHT_APPLIED;
   END_IF;
   #HMI_STANDARD.HMI_START_CONDITIONS := "M_ONE" AND #DATA_SEQUENCE.START_GENERAL_CONDITIONS AND #DATA_SEQUENCE.START_INITIAL_CONDITIONS;
   #HMI_STANDARD.HMI_STOP_CONDITIONS := "M_ONE" AND #DATA_SEQUENCE.STOP_GENERAL_CONDITIONS AND #DATA_SEQUENCE.STOP_INITIAL_CONDITIONS;
END_REGION

REGION Network 46: OUTPUTS
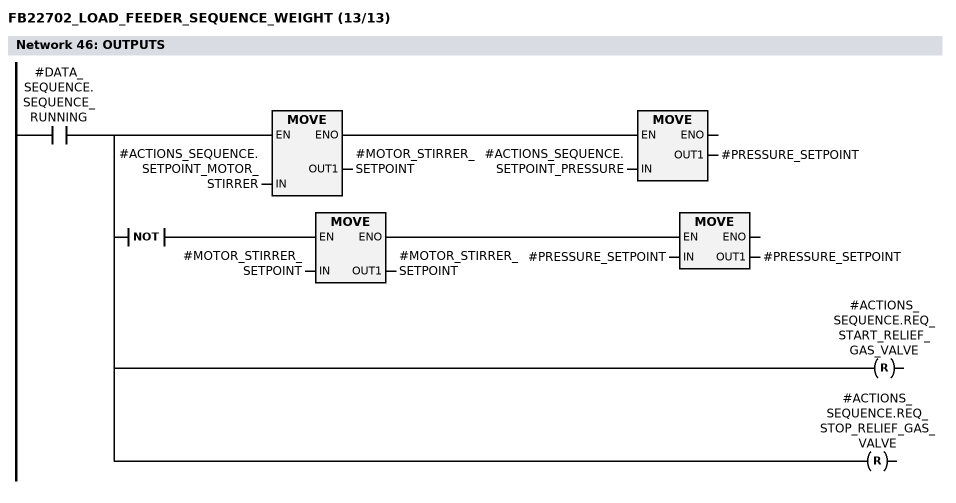
   RUNG wire#powerrail
      Contact( #DATA_SEQUENCE.SEQUENCE_RUNNING )
      wire#w1
      Move(in := #ACTIONS_SEQUENCE.SETPOINT_MOTOR_STIRRER, out1 => #MOTOR_STIRRER_SETPOINT)
      Move(in := #ACTIONS_SEQUENCE.SETPOINT_PRESSURE, out1 => #PRESSURE_SETPOINT)
   END_RUNG
   RUNG wire#w1
      Not()
      Move(in := #MOTOR_STIRRER_SETPOINT, out1 => #MOTOR_STIRRER_SETPOINT)
      Move(in := #PRESSURE_SETPOINT, out1 => #PRESSURE_SETPOINT)
   END_RUNG
   RUNG wire#w1
      R_Coil( #ACTIONS_SEQUENCE.REQ_START_RELIEF_GAS_VALVE )
   END_RUNG
   RUNG wire#w1
      R_Coil( #ACTIONS_SEQUENCE.REQ_STOP_RELIEF_GAS_VALVE )
   END_RUNG
   // the same network as SCL:
   IF #DATA_SEQUENCE.SEQUENCE_RUNNING THEN
       #MOTOR_STIRRER_SETPOINT := #ACTIONS_SEQUENCE.SETPOINT_MOTOR_STIRRER;
       #PRESSURE_SETPOINT := #ACTIONS_SEQUENCE.SETPOINT_PRESSURE;
   END_IF;
   IF NOT #DATA_SEQUENCE.SEQUENCE_RUNNING THEN
       #MOTOR_STIRRER_SETPOINT := #MOTOR_STIRRER_SETPOINT;
       #PRESSURE_SETPOINT := #PRESSURE_SETPOINT;
   END_IF;
   IF #DATA_SEQUENCE.SEQUENCE_RUNNING THEN
       #ACTIONS_SEQUENCE.REQ_START_RELIEF_GAS_VALVE := FALSE;
       #ACTIONS_SEQUENCE.REQ_STOP_RELIEF_GAS_VALVE := FALSE;
   END_IF;
END_REGION
END_FUNCTION_BLOCK
